C03648=1159.072,-127.448,-41.821,178.641,5.854,149.447
C03649=1159.067,-127.198,-41.829,178.642,5.854,149.447
C03650=1159.061,-126.949,-41.837,178.645,5.855,149.446
C03651=1159.055,-126.699,-41.846,178.646,5.855,149.446
C03652=1159.050,-126.448,-41.854,178.649,5.855,149.445
C03653=1159.045,-126.199,-41.862,178.651,5.855,149.445
C03654=1159.040,-125.950,-41.871,178.653,5.856,149.444
C03655=1159.034,-125.699,-41.879,178.654,5.856,149.444
C03656=1159.029,-125.450,-41.888,178.657,5.856,149.443
C03657=1159.023,-125.200,-41.897,178.659,5.856,149.443
C03658=1159.018,-124.950,-41.906,178.661,5.857,149.442
C03659=1159.013,-124.700,-41.914,178.662,5.857,149.442
C03660=1159.007,-124.451,-41.922,178.665,5.858,149.441
C03661=1159.002,-124.201,-41.931,178.666,5.857,149.441
C03662=1158.996,-123.950,-41.939,178.669,5.858,149.440
C03663=1158.991,-123.701,-41.947,178.670,5.858,149.439
C03664=1158.986,-123.452,-41.956,178.673,5.859,149.439
C03665=1158.981,-123.202,-41.965,178.674,5.859,149.438
C03666=1158.975,-122.952,-41.973,178.676,5.859,149.438
C03667=1158.970,-122.702,-41.982,178.679,5.859,149.437
C03668=1158.965,-122.452,-41.991,178.681,5.860,149.437
C03669=1158.959,-122.202,-42.000,178.682,5.860,149.436
C03670=1158.953,-121.953,-42.008,178.685,5.860,149.436
C03671=1158.948,-121.703,-42.016,178.686,5.860,149.435
C03672=1158.943,-121.453,-42.025,178.689,5.861,149.435
C03673=1158.938,-121.203,-42.034,178.690,5.861,149.434
C03674=1158.932,-120.953,-42.042,178.693,5.861,149.434
C03675=1158.927,-120.703,-42.051,178.694,5.861,149.433
C03676=1158.921,-120.454,-42.060,178.696,5.862,149.433
C03677=1158.916,-120.204,-42.069,178.698,5.862,149.432
C03678=1158.910,-119.955,-42.077,178.701,5.862,149.431
C03679=1158.905,-119.704,-42.085,178.702,5.862,149.431
C03680=1158.900,-119.454,-42.094,178.704,5.863,149.430
C03681=1158.895,-119.204,-42.103,178.707,5.863,149.430
C03682=1158.889,-118.955,-42.112,178.709,5.863,149.429
C03683=1158.884,-118.705,-42.121,178.710,5.863,149.429
C03684=1158.879,-118.456,-42.130,178.713,5.864,149.428
C03685=1158.873,-118.206,-42.138,178.715,5.865,149.428
C03686=1158.868,-117.955,-42.147,178.717,5.865,149.427
C03687=1158.862,-117.706,-42.155,178.719,5.865,149.427
C03688=1158.857,-117.456,-42.164,178.721,5.865,149.426
C03689=1158.852,-117.206,-42.173,178.723,5.866,149.426
C03690=1158.847,-116.957,-42.182,178.725,5.866,149.425
C03691=1158.841,-116.707,-42.190,178.727,5.866,149.424
C03692=1158.836,-116.458,-42.199,178.729,5.866,149.424
C03693=1158.831,-116.208,-42.208,178.731,5.867,149.423
C03694=1158.825,-115.958,-42.217,178.733,5.867,149.423
C03695=1158.820,-115.707,-42.225,178.735,5.867,149.422
C03696=1158.814,-115.458,-42.234,178.737,5.867,149.422
C03697=1158.808,-115.208,-42.243,178.739,5.868,149.421
C03698=1158.803,-114.958,-42.252,178.741,5.868,149.421
C03699=1158.798,-114.708,-42.261,178.743,5.868,149.420
C03700=1158.793,-114.458,-42.270,178.745,5.869,149.420
C03701=1158.788,-114.209,-42.279,178.747,5.869,149.419
C03702=1158.782,-113.959,-42.287,178.750,5.870,149.418
C03703=1158.777,-113.710,-42.296,178.751,5.869,149.418
C03704=1158.771,-113.460,-42.305,178.753,5.870,149.417
C03705=1158.766,-113.210,-42.314,178.755,5.870,149.417
C03706=1158.760,-112.960,-42.324,178.758,5.871,149.416
C03707=1158.755,-112.710,-42.333,178.759,5.871,149.416
C03708=1158.749,-112.461,-42.341,178.762,5.871,149.415
C03709=1158.744,-112.211,-42.350,178.763,5.871,149.415
C03710=1158.739,-111.961,-42.359,178.766,5.872,149.414
C03711=1158.734,-111.711,-42.368,178.768,5.872,149.414
C03712=1158.729,-111.461,-42.377,178.770,5.872,149.413
C03713=1158.723,-111.211,-42.386,178.772,5.873,149.413
C03714=1158.718,-110.961,-42.395,178.774,5.873,149.412
C03715=1158.712,-110.712,-42.404,178.776,5.873,149.411
C03716=1158.707,-110.462,-42.412,178.778,5.873,149.411
C03717=1158.702,-110.213,-42.421,178.780,5.874,149.410
C03718=1158.696,-109.963,-42.430,178.782,5.874,149.410
C03719=1158.691,-109.712,-42.440,178.784,5.875,149.409
C03720=1158.686,-109.463,-42.449,178.786,5.875,149.409
C03721=1158.681,-109.213,-42.458,178.788,5.875,149.408
C03722=1158.675,-108.964,-42.467,178.791,5.876,149.408
C03723=1158.670,-108.714,-42.476,178.792,5.876,149.407
C03724=1158.664,-108.464,-42.485,178.794,5.876,149.407
C03725=1158.659,-108.214,-42.494,178.796,5.876,149.406
C03726=1158.653,-107.965,-42.503,178.799,5.877,149.405
C03727=1158.648,-107.715,-42.512,178.801,5.877,149.405
C03728=1158.643,-107.465,-42.521,178.802,5.877,149.404
C03729=1158.637,-107.215,-42.531,178.805,5.878,149.404
C03730=1158.632,-106.965,-42.540,178.807,5.878,149.403
C03731=1158.627,-106.716,-42.549,178.809,5.879,149.403
C03732=1158.622,-106.466,-42.558,178.811,5.878,149.402
C03733=1158.616,-106.216,-42.567,178.813,5.879,149.401
C03734=1158.611,-105.966,-42.576,178.815,5.880,149.401
C03735=1158.606,-105.716,-42.586,178.817,5.880,149.401
C03736=1158.600,-105.467,-42.594,178.820,5.880,149.400
C03737=1158.594,-105.217,-42.604,178.821,5.880,149.399
C03738=1158.589,-104.967,-42.613,178.823,5.881,149.399
C03739=1158.584,-104.717,-42.622,178.826,5.880,149.398
C03740=1158.579,-104.468,-42.631,178.828,5.881,149.398
C03741=1158.573,-104.218,-42.641,178.830,5.882,149.397
C03742=1158.568,-103.968,-42.650,178.832,5.881,149.396
C03743=1158.563,-103.718,-42.658,178.834,5.882,149.396
C03744=1158.557,-103.469,-42.669,178.836,5.882,149.395
C03745=1158.552,-103.219,-42.678,178.838,5.883,149.395
C03746=1158.547,-102.969,-42.686,178.840,5.882,149.394
C03747=1158.541,-102.697,-42.697,178.842,5.883,149.394
C03748=1158.535,-102.425,-42.707,178.845,5.884,149.393
C03749=1158.529,-102.152,-42.717,178.847,5.884,149.393
C03750=1158.523,-101.881,-42.727,178.849,5.884,149.392
C03751=1158.518,-101.631,-42.736,178.851,5.885,149.391
C03752=1158.513,-101.382,-42.746,178.854,5.885,149.391
C03753=1158.507,-101.132,-42.755,178.856,5.885,149.390
C03754=1158.502,-100.882,-42.764,178.858,5.886,149.390
C03755=1158.497,-100.633,-42.774,178.859,5.886,149.389
C03756=1158.491,-100.383,-42.783,178.862,5.886,149.388
C03757=1158.486,-100.133,-42.792,178.864,5.887,149.388
C03758=1158.481,-99.883,-42.802,178.866,5.887,149.388
C03759=1158.476,-99.633,-42.811,178.869,5.887,149.387
C03760=1158.470,-99.384,-42.820,178.870,5.887,149.386
C03761=1158.465,-99.134,-42.830,178.872,5.888,149.386
C03762=1158.460,-98.884,-42.839,178.875,5.888,149.385
C03763=1158.454,-98.634,-42.848,178.877,5.888,149.385
C03764=1158.449,-98.385,-42.858,178.879,5.889,149.384
C03765=1158.444,-98.135,-42.867,178.881,5.889,149.383
C03766=1158.439,-97.885,-42.877,178.883,5.889,149.383
C03767=1158.434,-97.635,-42.886,178.885,5.890,149.382
C03768=1158.428,-97.385,-42.896,178.887,5.890,149.382
C03769=1158.423,-97.135,-42.905,178.890,5.891,149.381
C03770=1158.417,-96.885,-42.915,178.891,5.891,149.381
C03771=1158.412,-96.636,-42.925,178.893,5.891,149.380
C03772=1158.407,-96.386,-42.933,178.896,5.892,149.380
C03773=1158.401,-96.136,-42.943,178.898,5.892,149.379
C03774=1158.396,-95.887,-42.953,178.900,5.892,149.379
C03775=1158.390,-95.637,-42.962,178.903,5.893,149.378
C03776=1158.385,-95.387,-42.972,178.904,5.893,149.377
C03777=1158.379,-95.137,-42.981,178.906,5.894,149.377
C03778=1158.375,-94.888,-42.991,178.908,5.893,149.376
C03779=1158.369,-94.638,-43.000,178.911,5.894,149.376
C03780=1158.364,-94.389,-43.010,178.913,5.895,149.375
C03781=1158.358,-94.139,-43.019,178.915,5.894,149.375
C03782=1158.354,-93.889,-43.029,178.917,5.895,149.374
C03783=1158.348,-93.638,-43.039,178.920,5.895,149.373
C03784=1158.343,-93.389,-43.048,178.921,5.895,149.373
C03785=1158.337,-93.139,-43.058,178.924,5.896,149.372
C03786=1158.332,-92.890,-43.068,178.926,5.896,149.372
C03787=1158.326,-92.640,-43.077,178.928,5.897,149.371
C03788=1158.321,-92.390,-43.087,178.930,5.897,149.371
C03789=1158.315,-92.140,-43.096,178.932,5.897,149.370
C03790=1158.311,-91.891,-43.106,178.934,5.898,149.370
C03791=1158.305,-91.641,-43.115,178.936,5.898,149.369
C03792=1158.300,-91.391,-43.125,178.939,5.898,149.368
C03793=1158.294,-91.141,-43.135,178.941,5.899,149.368
C03794=1158.290,-90.892,-43.144,178.943,5.900,149.367
C03795=1158.284,-90.642,-43.155,178.945,5.899,149.367
C03796=1158.279,-90.392,-43.163,178.947,5.900,149.366
C03797=1158.273,-90.143,-43.174,178.949,5.900,149.366
C03798=1158.268,-89.893,-43.183,178.951,5.900,149.365
C03799=1158.263,-89.642,-43.193,178.954,5.901,149.364
C03800=1158.257,-89.393,-43.203,178.955,5.901,149.364
C03801=1158.252,-89.143,-43.212,178.958,5.901,149.363
C03802=1158.247,-88.894,-43.222,178.960,5.902,149.363
C03803=1158.242,-88.644,-43.232,178.962,5.902,149.362
C03804=1158.236,-88.394,-43.242,178.964,5.903,149.362
C03805=1158.231,-88.144,-43.252,178.967,5.903,149.361
C03806=1158.226,-87.894,-43.261,178.969,5.903,149.360
C03807=1158.220,-87.645,-43.271,178.971,5.904,149.360
C03808=1158.215,-87.395,-43.281,178.973,5.904,149.359
C03809=1158.209,-87.145,-43.290,178.975,5.904,149.359
C03810=1158.204,-86.896,-43.301,178.977,5.905,149.358
C03811=1158.200,-86.646,-43.311,178.980,5.905,149.358
C03812=1158.194,-86.396,-43.321,178.982,5.905,149.357
C03813=1158.189,-86.146,-43.330,178.984,5.906,149.357
C03814=1158.183,-85.897,-43.340,178.986,5.906,149.356
C03815=1158.178,-85.647,-43.350,178.988,5.906,149.355
C03816=1158.173,-85.397,-43.359,178.990,5.907,149.355
C03817=1158.167,-85.147,-43.370,178.992,5.907,149.354
C03818=1158.162,-84.898,-43.380,178.994,5.907,149.354
C03819=1158.157,-84.648,-43.389,178.997,5.908,149.353
C03820=1158.151,-84.398,-43.399,178.999,5.908,149.353
C03821=1158.146,-84.148,-43.409,179.001,5.909,149.352
C03822=1158.141,-83.899,-43.419,179.004,5.909,149.351
C03823=1158.136,-83.649,-43.429,179.006,5.910,149.351
C03824=1158.130,-83.399,-43.439,179.007,5.910,149.350
C03825=1158.125,-83.149,-43.449,179.010,5.910,149.350
C03826=1158.120,-82.899,-43.459,179.012,5.911,149.349
C03827=1158.114,-82.650,-43.469,179.014,5.910,149.348
C03828=1158.109,-82.400,-43.479,179.017,5.911,149.348
C03829=1158.104,-82.150,-43.489,179.019,5.912,149.348
C03830=1158.099,-81.900,-43.499,179.021,5.912,149.347
C03831=1158.093,-81.651,-43.509,179.023,5.912,149.346
C03832=1158.088,-81.402,-43.519,179.025,5.913,149.346
C03833=1158.083,-81.151,-43.529,179.027,5.913,149.345
C03834=1158.077,-80.902,-43.539,179.029,5.913,149.345
C03835=1158.072,-80.652,-43.550,179.032,5.914,149.344
C03836=1158.067,-80.402,-43.559,179.034,5.914,149.343
C03837=1158.062,-80.152,-43.569,179.036,5.915,149.343
C03838=1158.056,-79.903,-43.579,179.039,5.915,149.342
C03839=1158.050,-79.653,-43.590,179.040,5.915,149.342
C03840=1158.046,-79.403,-43.600,179.043,5.915,149.341
C03841=1158.041,-79.154,-43.610,179.045,5.916,149.341
C03842=1158.035,-78.904,-43.620,179.047,5.916,149.340
C03843=1158.029,-78.654,-43.630,179.049,5.917,149.339
C03844=1158.024,-78.404,-43.641,179.051,5.917,149.339
C03845=1158.019,-78.154,-43.650,179.054,5.918,149.338
C03846=1158.014,-77.905,-43.660,179.056,5.918,149.338
C03847=1158.009,-77.655,-43.670,179.058,5.918,149.337
C03848=1158.003,-77.405,-43.681,179.061,5.919,149.337
C03849=1157.997,-77.155,-43.691,179.062,5.919,149.336
C03850=1157.992,-76.906,-43.701,179.065,5.919,149.335
C03851=1157.987,-76.635,-43.712,179.067,5.920,149.335
C03852=1157.981,-76.363,-43.724,179.070,5.920,149.334
C03853=1157.976,-76.092,-43.734,179.072,5.921,149.334
C03854=1157.969,-75.821,-43.746,179.074,5.921,149.333
C03855=1157.965,-75.571,-43.756,179.076,5.922,149.332
C03856=1157.959,-75.321,-43.766,179.079,5.922,149.332
C03857=1157.954,-75.072,-43.776,179.081,5.923,149.331
C03858=1157.949,-74.822,-43.787,179.083,5.922,149.331
C03859=1157.943,-74.572,-43.797,179.085,5.923,149.330
C03860=1157.937,-74.322,-43.807,179.088,5.923,149.329
C03861=1157.932,-74.072,-43.818,179.090,5.923,149.329
C03862=1157.927,-73.823,-43.828,179.092,5.924,149.328
C03863=1157.921,-73.573,-43.838,179.094,5.925,149.328
C03864=1157.917,-73.323,-43.848,179.097,5.925,149.327
C03865=1157.911,-73.074,-43.858,179.099,5.925,149.327
C03866=1157.906,-72.824,-43.868,179.101,5.926,149.326
C03867=1157.901,-72.574,-43.880,179.103,5.927,149.326
C03868=1157.895,-72.325,-43.890,179.105,5.926,149.325
C03869=1157.890,-72.075,-43.900,179.107,5.927,149.324
C03870=1157.885,-71.825,-43.911,179.110,5.927,149.324
C03871=1157.879,-71.576,-43.921,179.112,5.928,149.323
C03872=1157.874,-71.325,-43.931,179.114,5.928,149.322
C03873=1157.869,-71.076,-43.942,179.117,5.928,149.322
C03874=1157.863,-70.826,-43.952,179.119,5.929,149.322
C03875=1157.858,-70.576,-43.962,179.121,5.930,149.321
C03876=1157.853,-70.327,-43.973,179.123,5.930,149.320
C03877=1157.848,-70.077,-43.984,179.126,5.930,149.320
C03878=1157.842,-69.827,-43.994,179.128,5.931,149.319
C03879=1157.837,-69.577,-44.005,179.131,5.931,149.318
C03880=1157.832,-69.328,-44.015,179.132,5.931,149.318
C03881=1157.826,-69.078,-44.025,179.134,5.932,149.317
C03882=1157.821,-68.828,-44.036,179.137,5.932,149.317
C03883=1157.816,-68.579,-44.047,179.139,5.932,149.316
C03884=1157.811,-68.329,-44.057,179.141,5.933,149.316
C03885=1157.805,-68.079,-44.067,179.143,5.933,149.315
C03886=1157.800,-67.829,-44.078,179.146,5.934,149.314
C03887=1157.795,-67.580,-44.089,179.148,5.934,149.314
C03888=1157.789,-67.330,-44.099,179.150,5.935,149.313
C03889=1157.784,-67.080,-44.110,179.153,5.935,149.313
C03890=1157.779,-66.831,-44.120,179.155,5.936,149.312
C03891=1157.774,-66.581,-44.131,179.157,5.935,149.312
C03892=1157.768,-66.331,-44.141,179.159,5.936,149.311
C03893=1157.763,-66.081,-44.152,179.162,5.937,149.310
C03894=1157.758,-65.832,-44.162,179.164,5.937,149.310
C03895=1157.753,-65.582,-44.173,179.165,5.937,149.309
C03896=1157.747,-65.332,-44.184,179.168,5.938,149.309
C03897=1157.742,-65.082,-44.194,179.170,5.939,149.308
C03898=1157.737,-64.833,-44.205,179.173,5.939,149.307
C03899=1157.732,-64.583,-44.216,179.175,5.940,149.307
C03900=1157.727,-64.333,-44.226,179.177,5.939,149.306
C03901=1157.722,-64.084,-44.237,179.179,5.940,149.306
C03902=1157.716,-63.834,-44.247,179.182,5.941,149.305
C03903=1157.711,-63.584,-44.258,179.184,5.941,149.305
C03904=1157.705,-63.335,-44.270,179.186,5.941,149.304
C03905=1157.700,-63.085,-44.280,179.189,5.942,149.303
C03906=1157.695,-62.835,-44.290,179.191,5.942,149.303
C03907=1157.690,-62.585,-44.302,179.193,5.943,149.302
C03908=1157.684,-62.336,-44.312,179.195,5.943,149.302
C03909=1157.679,-62.086,-44.322,179.198,5.943,149.301
C03910=1157.674,-61.837,-44.333,179.200,5.944,149.301
C03911=1157.669,-61.586,-44.344,179.203,5.944,149.300
C03912=1157.663,-61.337,-44.355,179.205,5.945,149.299
C03913=1157.658,-61.087,-44.366,179.206,5.945,149.299
C03914=1157.652,-60.837,-44.376,179.209,5.946,149.298
C03915=1157.648,-60.588,-44.388,179.211,5.946,149.298
C03916=1157.643,-60.338,-44.398,179.214,5.947,149.297
C03917=1157.637,-60.089,-44.409,179.215,5.947,149.297
C03918=1157.632,-59.838,-44.420,179.218,5.947,149.296
C03919=1157.626,-59.589,-44.431,179.220,5.948,149.295
C03920=1157.621,-59.339,-44.442,179.223,5.948,149.295
C03921=1157.616,-59.090,-44.453,179.225,5.949,149.294
C03922=1157.611,-58.840,-44.463,179.227,5.949,149.294
C03923=1157.606,-58.590,-44.474,179.229,5.950,149.293
C03924=1157.600,-58.340,-44.485,179.232,5.950,149.293
C03925=1157.595,-58.091,-44.497,179.234,5.951,149.292
C03926=1157.590,-57.841,-44.507,179.236,5.952,149.291
C03927=1157.585,-57.591,-44.518,179.238,5.951,149.291
C03928=1157.580,-57.341,-44.529,179.241,5.952,149.290
C03929=1157.574,-57.092,-44.540,179.243,5.952,149.289
C03930=1157.569,-56.842,-44.551,179.246,5.953,149.289
C03931=1157.564,-56.593,-44.562,179.248,5.954,149.288
C03932=1157.559,-56.343,-44.572,179.250,5.954,149.288
C03933=1157.553,-56.093,-44.584,179.252,5.954,149.287
C03934=1157.548,-55.844,-44.595,179.255,5.955,149.287
C03935=1157.543,-55.593,-44.606,179.257,5.955,149.286
C03936=1157.538,-55.345,-44.617,179.260,5.956,149.285
C03937=1157.532,-55.094,-44.628,179.261,5.956,149.285
C03938=1157.527,-54.844,-44.639,179.264,5.956,149.284
C03939=1157.522,-54.595,-44.649,179.266,5.957,149.284
C03940=1157.517,-54.345,-44.661,179.269,5.957,149.283
C03941=1157.512,-54.095,-44.672,179.271,5.958,149.283
C03942=1157.506,-53.846,-44.683,179.273,5.958,149.282
C03943=1157.501,-53.596,-44.694,179.275,5.959,149.281
C03944=1157.496,-53.346,-44.706,179.278,5.959,149.281
C03945=1157.490,-53.097,-44.716,179.280,5.960,149.280
C03946=1157.486,-52.847,-44.727,179.283,5.960,149.280
C03947=1157.480,-52.597,-44.739,179.284,5.960,149.279
C03948=1157.475,-52.347,-44.749,179.287,5.961,149.278
C03949=1157.470,-52.098,-44.761,179.289,5.961,149.278
C03950=1157.465,-51.848,-44.773,179.292,5.962,149.277
C03951=1157.459,-51.598,-44.783,179.294,5.963,149.277
C03952=1157.454,-51.349,-44.794,179.296,5.963,149.276
C03953=1157.449,-51.099,-44.806,179.298,5.963,149.276
C03954=1157.443,-50.849,-44.816,179.300,5.964,149.275
C03955=1157.438,-50.579,-44.829,179.303,5.964,149.274
C03956=1157.432,-50.308,-44.841,179.306,5.965,149.274
C03957=1157.426,-50.038,-44.853,179.308,5.965,149.273
C03958=1157.421,-49.767,-44.865,179.311,5.966,149.272
C03959=1157.416,-49.517,-44.877,179.313,5.966,149.272
C03960=1157.410,-49.268,-44.888,179.315,5.967,149.271
C03961=1157.405,-49.018,-44.899,179.318,5.967,149.271
C03962=1157.400,-48.768,-44.910,179.320,5.968,149.270
C03963=1157.395,-48.519,-44.921,179.322,5.968,149.269
C03964=1157.389,-48.269,-44.933,179.324,5.969,149.269
C03965=1157.385,-48.019,-44.944,179.327,5.969,149.268
C03966=1157.379,-47.769,-44.955,179.329,5.970,149.268
C03967=1157.374,-47.520,-44.966,179.332,5.971,149.267
C03968=1157.368,-47.270,-44.978,179.334,5.971,149.267
C03969=1157.363,-47.020,-44.990,179.336,5.971,149.266
C03970=1157.357,-46.771,-45.001,179.338,5.971,149.265
C03971=1157.353,-46.522,-45.012,179.341,5.972,149.265
C03972=1157.347,-46.271,-45.024,179.343,5.973,149.264
C03973=1157.342,-46.021,-45.035,179.345,5.973,149.264
C03974=1157.338,-45.772,-45.046,179.348,5.974,149.263
C03975=1157.332,-45.523,-45.058,179.350,5.975,149.263
C03976=1157.327,-45.273,-45.069,179.352,5.974,149.262
C03977=1157.321,-45.023,-45.081,179.355,5.975,149.261
C03978=1157.317,-44.773,-45.092,179.357,5.975,149.261
C03979=1157.311,-44.524,-45.104,179.359,5.976,149.260
C03980=1157.306,-44.274,-45.115,179.362,5.977,149.259
C03981=1157.301,-44.025,-45.127,179.364,5.977,149.259
C03982=1157.296,-43.774,-45.137,179.367,5.978,149.258
C03983=1157.290,-43.524,-45.149,179.369,5.979,149.258
C03984=1157.284,-43.275,-45.161,179.371,5.978,149.257
C03985=1157.279,-43.025,-45.172,179.373,5.979,149.257
C03986=1157.274,-42.776,-45.184,179.376,5.979,149.256
C03987=1157.269,-42.526,-45.195,179.378,5.980,149.255
C03988=1157.264,-42.276,-45.207,179.381,5.981,149.255
C03989=1157.259,-42.027,-45.218,179.383,5.981,149.254
C03990=1157.253,-41.777,-45.230,179.386,5.982,149.254
C03991=1157.248,-41.528,-45.241,179.388,5.983,149.253
C03992=1157.243,-41.278,-45.253,179.390,5.982,149.252
C03993=1157.238,-41.028,-45.265,179.392,5.983,149.252
C03994=1157.232,-40.779,-45.276,179.395,5.984,149.251
C03995=1157.227,-40.529,-45.288,179.397,5.984,149.251
C03996=1157.222,-40.279,-45.299,179.400,5.985,149.250
C03997=1157.217,-40.029,-45.311,179.402,5.986,149.250
C03998=1157.211,-39.779,-45.323,179.405,5.986,149.249
C03999=1157.207,-39.530,-45.334,179.407,5.987,149.248
C04000=1157.202,-39.280,-45.347,179.409,5.986,149.248
C04001=1157.196,-39.031,-45.358,179.411,5.987,149.247
C04002=1157.191,-38.781,-45.370,179.413,5.988,149.247
C04003=1157.185,-38.532,-45.381,179.416,5.988,149.246
C04004=1157.181,-38.282,-45.393,179.418,5.989,149.246
C04005=1157.175,-38.032,-45.405,179.421,5.990,149.245
C04006=1157.170,-37.782,-45.416,179.423,5.990,149.244
C04007=1157.165,-37.532,-45.428,179.426,5.991,149.244
C04008=1157.159,-37.283,-45.439,179.428,5.992,149.243
C04009=1157.154,-37.033,-45.451,179.430,5.992,149.243
C04010=1157.149,-36.784,-45.463,179.432,5.992,149.242
C04011=1157.144,-36.534,-45.475,179.435,5.992,149.241
C04012=1157.138,-36.284,-45.487,179.437,5.993,149.241
C04013=1157.134,-36.035,-45.498,179.439,5.994,149.240
C04014=1157.128,-35.785,-45.510,179.442,5.994,149.240
C04015=1157.123,-35.535,-45.522,179.444,5.995,149.239
C04016=1157.119,-35.286,-45.534,179.447,5.996,149.239
C04017=1157.113,-35.036,-45.546,179.449,5.996,149.238
C04018=1157.107,-34.787,-45.557,179.451,5.997,149.237
C04019=1157.102,-34.537,-45.569,179.454,5.997,149.237
C04020=1157.097,-34.288,-45.581,179.456,5.998,149.236
C04021=1157.092,-34.038,-45.593,179.458,5.998,149.236
C04022=1157.086,-33.788,-45.605,179.460,5.999,149.235
C04023=1157.081,-33.538,-45.617,179.463,5.999,149.234
C04024=1157.077,-33.289,-45.629,179.465,6.000,149.234
C04025=1157.071,-33.039,-45.641,179.468,6.000,149.233
C04026=1157.066,-32.789,-45.653,179.470,6.001,149.233
C04027=1157.060,-32.539,-45.665,179.473,6.001,149.232
C04028=1157.056,-32.290,-45.677,179.475,6.002,149.232
C04029=1157.050,-32.040,-45.689,179.478,6.003,149.231
C04030=1157.045,-31.790,-45.700,179.480,6.003,149.230
C04031=1157.040,-31.541,-45.713,179.483,6.004,149.230
C04032=1157.034,-31.291,-45.725,179.485,6.005,149.229
C04033=1157.030,-31.041,-45.736,179.487,6.005,149.228
C04034=1157.024,-30.791,-45.748,179.490,6.006,149.228
C04035=1157.019,-30.542,-45.761,179.492,6.005,149.227
C04036=1157.014,-30.292,-45.773,179.494,6.006,149.227
C04037=1157.009,-30.043,-45.785,179.496,6.007,149.226
C04038=1157.004,-29.793,-45.796,179.499,6.007,149.225
C04039=1156.999,-29.543,-45.808,179.501,6.008,149.225
C04040=1156.993,-29.294,-45.821,179.504,6.008,149.224
C04041=1156.988,-29.044,-45.833,179.506,6.009,149.224
C04042=1156.983,-28.794,-45.845,179.509,6.010,149.223
C04043=1156.977,-28.545,-45.857,179.511,6.010,149.223
C04044=1156.972,-28.295,-45.869,179.514,6.011,149.222
C04045=1156.968,-28.046,-45.881,179.516,6.012,149.221
C04046=1156.962,-27.796,-45.893,179.518,6.012,149.221
C04047=1156.957,-27.547,-45.906,179.521,6.013,149.220
C04048=1156.952,-27.297,-45.918,179.523,6.013,149.220
C04049=1156.946,-27.047,-45.929,179.526,6.014,149.219
C04050=1156.941,-26.797,-45.942,179.528,6.014,149.218
C04051=1156.936,-26.547,-45.954,179.530,6.015,149.218
C04052=1156.931,-26.298,-45.967,179.533,6.016,149.217
C04053=1156.926,-26.049,-45.978,179.535,6.016,149.217
C04054=1156.921,-25.799,-45.990,179.538,6.017,149.216
C04055=1156.915,-25.549,-46.002,179.540,6.018,149.216
C04056=1156.910,-25.300,-46.015,179.543,6.018,149.215
C04057=1156.905,-25.050,-46.027,179.544,6.018,149.214
C04058=1156.900,-24.800,-46.040,179.547,6.019,149.214
C04059=1156.894,-24.530,-46.052,179.550,6.020,149.213
C04060=1156.889,-24.260,-46.067,179.552,6.021,149.213
C04061=1156.883,-23.991,-46.079,179.555,6.021,149.212
C04062=1156.878,-23.721,-46.093,179.558,6.021,149.211
C04063=1156.872,-23.471,-46.105,179.560,6.022,149.211
C04064=1156.867,-23.222,-46.117,179.563,6.023,149.210
C04065=1156.862,-22.972,-46.129,179.565,6.023,149.210
C04066=1156.857,-22.722,-46.142,179.567,6.024,149.209
C04067=1156.852,-22.472,-46.154,179.570,6.025,149.208
C04068=1156.847,-22.222,-46.167,179.572,6.025,149.208
C04069=1156.841,-21.973,-46.179,179.574,6.026,149.207
C04070=1156.836,-21.723,-46.191,179.577,6.026,149.207
C04071=1156.831,-21.474,-46.204,179.579,6.027,149.206
C04072=1156.826,-21.225,-46.216,179.582,6.028,149.205
C04073=1156.820,-20.975,-46.228,179.584,6.028,149.205
C04074=1156.815,-20.725,-46.241,179.587,6.029,149.204
C04075=1156.811,-20.475,-46.254,179.589,6.030,149.204
C04076=1156.805,-20.225,-46.266,179.592,6.030,149.203
C04077=1156.800,-19.976,-46.278,179.594,6.031,149.203
C04078=1156.794,-19.726,-46.292,179.596,6.031,149.202
C04079=1156.789,-19.476,-46.303,179.599,6.032,149.201
C04080=1156.784,-19.227,-46.316,179.601,6.033,149.201
C04081=1156.779,-18.978,-46.329,179.603,6.033,149.200
C04082=1156.774,-18.727,-46.341,179.606,6.034,149.200
C04083=1156.769,-18.478,-46.354,179.608,6.035,149.199
C04084=1156.764,-18.229,-46.366,179.611,6.035,149.198
C04085=1156.758,-17.979,-46.379,179.613,6.036,149.198
C04086=1156.753,-17.729,-46.391,179.616,6.036,149.197
C04087=1156.748,-17.479,-46.404,179.618,6.037,149.197
C04088=1156.743,-17.230,-46.416,179.621,6.037,149.196
C04089=1156.737,-16.980,-46.429,179.623,6.038,149.196
C04090=1156.732,-16.730,-46.441,179.625,6.039,149.195
C04091=1156.727,-16.481,-46.454,179.628,6.040,149.194
C04092=1156.722,-16.231,-46.467,179.630,6.040,149.194
C04093=1156.717,-15.982,-46.479,179.632,6.041,149.193
C04094=1156.712,-15.732,-46.492,179.635,6.041,149.193
C04095=1156.707,-15.482,-46.504,179.637,6.042,149.192
C04096=1156.701,-15.233,-46.517,179.640,6.042,149.191
C04097=1156.696,-14.983,-46.530,179.642,6.043,149.191
C04098=1156.691,-14.734,-46.543,179.645,6.044,149.190
C04099=1156.686,-14.484,-46.555,179.647,6.044,149.190
C04100=1156.681,-14.235,-46.568,179.650,6.045,149.189
C04101=1156.676,-13.985,-46.581,179.652,6.045,149.188
C04102=1156.670,-13.735,-46.593,179.655,6.046,149.188
C04103=1156.665,-13.485,-46.606,179.657,6.047,149.187
C04104=1156.660,-13.236,-46.619,179.659,6.047,149.187
C04105=1156.656,-12.986,-46.631,179.662,6.048,149.186
C04106=1156.650,-12.736,-46.645,179.664,6.049,149.186
C04107=1156.645,-12.487,-46.657,179.667,6.049,149.185
C04108=1156.639,-12.238,-46.670,179.669,6.050,149.184
C04109=1156.635,-11.988,-46.683,179.672,6.050,149.184
C04110=1156.630,-11.738,-46.695,179.674,6.051,149.183
C04111=1156.624,-11.489,-46.709,179.677,6.052,149.183
C04112=1156.619,-11.239,-46.721,179.679,6.053,149.182
C04113=1156.614,-10.989,-46.734,179.682,6.054,149.181
C04114=1156.609,-10.740,-46.747,179.684,6.054,149.181
C04115=1156.603,-10.490,-46.760,179.687,6.055,149.180
C04116=1156.599,-10.240,-46.773,179.689,6.056,149.180
C04117=1156.594,-9.991,-46.786,179.692,6.056,149.179
C04118=1156.588,-9.741,-46.799,179.694,6.057,149.179
C04119=1156.583,-9.491,-46.812,179.696,6.057,149.178
C04120=1156.578,-9.242,-46.824,179.699,6.058,149.177
C04121=1156.573,-8.993,-46.837,179.701,6.059,149.177
C04122=1156.568,-8.742,-46.850,179.703,6.059,149.176
C04123=1156.563,-8.493,-46.863,179.706,6.060,149.176
C04124=1156.557,-8.244,-46.876,179.708,6.061,149.175
C04125=1156.552,-7.994,-46.889,179.711,6.061,149.174
C04126=1156.547,-7.744,-46.902,179.713,6.062,149.174
C04127=1156.542,-7.495,-46.914,179.716,6.062,149.173
C04128=1156.537,-7.245,-46.928,179.719,6.064,149.173
C04129=1156.532,-6.995,-46.941,179.721,6.064,149.172
C04130=1156.527,-6.747,-46.954,179.723,6.065,149.172
C04131=1156.522,-6.496,-46.967,179.726,6.066,149.171
C04132=1156.516,-6.247,-46.980,179.729,6.066,149.170
C04133=1156.511,-5.997,-46.993,179.731,6.067,149.170
C04134=1156.506,-5.747,-47.006,179.734,6.067,149.169
C04135=1156.501,-5.498,-47.019,179.736,6.068,149.169
C04136=1156.496,-5.248,-47.032,179.738,6.069,149.168
C04137=1156.491,-4.999,-47.046,179.741,6.070,149.168
C04138=1156.485,-4.749,-47.059,179.743,6.070,149.167
C04139=1156.480,-4.499,-47.072,179.745,6.071,149.166
C04140=1156.475,-4.250,-47.084,179.748,6.071,149.166
C04141=1156.469,-4.000,-47.098,179.751,6.073,149.165
C04142=1156.465,-3.751,-47.111,179.753,6.073,149.165
C04143=1156.459,-3.501,-47.125,179.756,6.074,149.164
C04144=1156.455,-3.251,-47.138,179.758,6.075,149.163
C04145=1156.449,-3.002,-47.151,179.760,6.075,149.163
C04146=1156.445,-2.752,-47.164,179.763,6.076,149.162
C04147=1156.440,-2.503,-47.177,179.765,6.077,149.162
C04148=1156.434,-2.253,-47.190,179.768,6.077,149.161
C04149=1156.429,-2.003,-47.203,179.770,6.078,149.161
C04150=1156.424,-1.754,-47.217,179.773,6.078,149.160
C04151=1156.419,-1.504,-47.230,179.776,6.080,149.159
C04152=1156.413,-1.255,-47.243,179.778,6.080,149.159
C04153=1156.409,-1.005,-47.257,179.780,6.081,149.158
C04154=1156.403,-0.756,-47.270,179.783,6.082,149.158
C04155=1156.398,-0.506,-47.283,179.785,6.082,149.157
C04156=1156.393,-0.257,-47.297,179.788,6.083,149.156
C04157=1156.388,-0.007,-47.310,179.790,6.084,149.156
C04158=1156.383,0.243,-47.323,179.793,6.084,149.155
C04159=1156.377,0.492,-47.337,179.795,6.085,149.155
C04160=1156.373,0.742,-47.350,179.798,6.086,149.154
C04161=1156.367,0.992,-47.363,179.800,6.087,149.154
C04162=1156.363,1.241,-47.377,179.803,6.087,149.153
C04163=1156.356,1.510,-47.391,179.806,6.088,149.152
C04164=1156.351,1.780,-47.406,179.808,6.089,149.152
C04165=1156.346,2.049,-47.420,179.811,6.090,149.151
C04166=1156.340,2.319,-47.435,179.814,6.090,149.150
C04167=1156.335,2.568,-47.448,179.816,6.091,149.150
C04168=1156.330,2.818,-47.461,179.818,6.092,149.149
C04169=1156.324,3.068,-47.475,179.821,6.093,149.149
C04170=1156.320,3.317,-47.489,179.823,6.093,149.148
C04171=1156.314,3.567,-47.501,179.826,6.095,149.148
C04172=1156.309,3.816,-47.516,179.829,6.095,149.147
C04173=1156.304,4.066,-47.528,179.831,6.096,149.147
C04174=1156.299,4.315,-47.543,179.834,6.096,149.146
C04175=1156.293,4.565,-47.556,179.836,6.097,149.145
C04176=1156.289,4.814,-47.569,179.838,6.098,149.145
C04177=1156.283,5.064,-47.583,179.841,6.098,149.144
C04178=1156.278,5.314,-47.597,179.844,6.100,149.144
C04179=1156.273,5.563,-47.610,179.846,6.100,149.143
C04180=1156.268,5.813,-47.624,179.849,6.101,149.142
C04181=1156.264,6.062,-47.638,179.851,6.102,149.142
C04182=1156.258,6.312,-47.651,179.853,6.102,149.141
C04183=1156.253,6.562,-47.665,179.856,6.103,149.141
C04184=1156.247,6.811,-47.678,179.858,6.103,149.140
C04185=1156.243,7.061,-47.692,179.862,6.105,149.139
C04186=1156.237,7.310,-47.705,179.864,6.106,149.139
C04187=1156.232,7.560,-47.719,179.866,6.106,149.138
C04188=1156.228,7.809,-47.733,179.869,6.107,149.138
C04189=1156.222,8.059,-47.746,179.871,6.107,149.137
C04190=1156.217,8.309,-47.760,179.873,6.108,149.137
C04191=1156.212,8.558,-47.773,179.877,6.109,149.136
C04192=1156.207,8.808,-47.787,179.879,6.110,149.136
C04193=1156.202,9.057,-47.802,179.881,6.111,149.135
C04194=1156.197,9.307,-47.815,179.884,6.111,149.134
C04195=1156.192,9.556,-47.829,179.886,6.112,149.134
C04196=1156.187,9.805,-47.842,179.888,6.113,149.133
C04197=1156.181,10.056,-47.856,179.892,6.114,149.133
C04198=1156.177,10.306,-47.870,179.894,6.115,149.132
C04199=1156.171,10.555,-47.884,179.896,6.115,149.131
C04200=1156.167,10.804,-47.898,179.899,6.116,149.131
C04201=1156.161,11.054,-47.911,179.901,6.117,149.130
C04202=1156.156,11.303,-47.925,179.904,6.118,149.130
C04203=1156.151,11.553,-47.940,179.907,6.119,149.129
C04204=1156.146,11.803,-47.953,179.909,6.119,149.129
C04205=1156.141,12.052,-47.967,179.912,6.120,149.128
C04206=1156.136,12.302,-47.981,179.914,6.121,149.128
C04207=1156.131,12.551,-47.995,179.916,6.121,149.127
C04208=1156.125,12.800,-48.009,179.919,6.123,149.126
C04209=1156.120,13.051,-48.023,179.922,6.123,149.126
C04210=1156.116,13.300,-48.036,179.924,6.124,149.125
C04211=1156.110,13.549,-48.050,179.927,6.125,149.125
C04212=1156.105,13.799,-48.064,179.929,6.125,149.124
C04213=1156.101,14.049,-48.079,179.932,6.127,149.123
C04214=1156.095,14.298,-48.092,179.934,6.127,149.123
C04215=1156.090,14.548,-48.106,179.937,6.128,149.122
C04216=1156.085,14.798,-48.120,179.939,6.129,149.122
C04217=1156.079,15.047,-48.134,179.942,6.129,149.121
C04218=1156.075,15.296,-48.148,179.944,6.131,149.121
C04219=1156.070,15.546,-48.162,179.947,6.131,149.120
C04220=1156.065,15.795,-48.177,179.949,6.132,149.120
C04221=1156.059,16.044,-48.190,179.952,6.133,149.119
C04222=1156.054,16.295,-48.204,179.954,6.133,149.118
C04223=1156.049,16.545,-48.218,179.957,6.135,149.118
C04224=1156.044,16.794,-48.232,179.959,6.136,149.117
C04225=1156.039,17.043,-48.247,179.962,6.136,149.117
C04226=1156.034,17.293,-48.261,179.964,6.137,149.116
C04227=1156.029,17.543,-48.275,179.968,6.138,149.115
C04228=1156.023,17.792,-48.289,179.970,6.139,149.115
C04229=1156.018,18.041,-48.303,179.972,6.139,149.114
C04230=1156.013,18.291,-48.318,179.975,6.140,149.114
C04231=1156.008,18.541,-48.332,179.977,6.141,149.113
C04232=1156.003,18.791,-48.346,179.980,6.142,149.113
C04233=1155.998,19.040,-48.360,179.983,6.143,149.112
C04234=1155.993,19.289,-48.374,179.985,6.144,149.112
C04235=1155.988,19.539,-48.389,179.987,6.144,149.111
C04236=1155.983,19.789,-48.403,179.990,6.146,149.110
C04237=1155.978,20.038,-48.417,179.993,6.146,149.110
C04238=1155.973,20.287,-48.431,179.995,6.147,149.109
C04239=1155.968,20.537,-48.445,179.998,6.147,149.109
C04240=1155.963,20.787,-48.460,-180.000,6.149,149.108
C04241=1155.958,21.037,-48.474,-179.997,6.149,149.107
C04242=1155.952,21.286,-48.488,-179.995,6.150,149.107
C04243=1155.947,21.535,-48.502,-179.992,6.151,149.106
C04244=1155.943,21.784,-48.517,-179.989,6.152,149.106
C04245=1155.938,22.034,-48.531,-179.987,6.153,149.105
C04246=1155.933,22.284,-48.546,-179.985,6.154,149.105
C04247=1155.928,22.533,-48.560,-179.982,6.154,149.104
C04248=1155.922,22.782,-48.574,-179.979,6.156,149.104
C04249=1155.917,23.032,-48.588,-179.977,6.156,149.103
C04250=1155.912,23.282,-48.602,-179.974,6.157,149.102
C04251=1155.907,23.532,-48.617,-179.972,6.158,149.102
C04252=1155.903,23.781,-48.632,-179.969,6.159,149.101
C04253=1155.897,24.031,-48.646,-179.966,6.160,149.101
C04254=1155.891,24.280,-48.660,-179.964,6.161,149.100
C04255=1155.886,24.529,-48.675,-179.961,6.161,149.100
C04256=1155.881,24.779,-48.689,-179.959,6.163,149.099
C04257=1155.877,25.028,-48.704,-179.956,6.163,149.098
C04258=1155.872,25.278,-48.718,-179.954,6.164,149.098
C04259=1155.867,25.528,-48.732,-179.951,6.164,149.097
C04260=1155.861,25.778,-48.747,-179.948,6.166,149.097
C04261=1155.857,26.027,-48.762,-179.946,6.166,149.096
C04262=1155.851,26.276,-48.776,-179.944,6.167,149.096
C04263=1155.846,26.525,-48.791,-179.941,6.169,149.095
C04264=1155.841,26.775,-48.805,-179.938,6.169,149.095
C04265=1155.836,27.024,-48.820,-179.936,6.170,149.094
C04266=1155.831,27.274,-48.835,-179.933,6.171,149.093
C04267=1155.826,27.543,-48.850,-179.930,6.172,149.093
C04268=1155.820,27.812,-48.866,-179.928,6.173,149.092
C04269=1155.815,28.081,-48.881,-179.925,6.174,149.092
C04270=1155.809,28.350,-48.897,-179.922,6.175,149.091
C04271=1155.805,28.599,-48.912,-179.919,6.176,149.090
C04272=1155.800,28.849,-48.927,-179.917,6.177,149.090
C04273=1155.795,29.099,-48.941,-179.915,6.178,149.089
C04274=1155.789,29.348,-48.956,-179.912,6.178,149.089
C04275=1155.784,29.597,-48.970,-179.909,6.180,149.088
C04276=1155.779,29.847,-48.985,-179.907,6.180,149.088
C04277=1155.773,30.096,-49.000,-179.904,6.181,149.087
C04278=1155.768,30.346,-49.015,-179.902,6.183,149.087
C04279=1155.764,30.595,-49.030,-179.899,6.183,149.086
C04280=1155.759,30.845,-49.044,-179.897,6.184,149.086
C04281=1155.753,31.094,-49.059,-179.894,6.185,149.085
C04282=1155.748,31.344,-49.074,-179.891,6.186,149.084
C04283=1155.743,31.594,-49.088,-179.889,6.186,149.084
C04284=1155.738,31.843,-49.104,-179.887,6.187,149.083
C04285=1155.733,32.093,-49.118,-179.883,6.189,149.083
C04286=1155.728,32.342,-49.133,-179.881,6.189,149.082
C04287=1155.724,32.592,-49.147,-179.879,6.190,149.081
C04288=1155.718,32.841,-49.163,-179.876,6.192,149.081
C04289=1155.713,33.091,-49.177,-179.873,6.192,149.080
C04290=1155.709,33.340,-49.192,-179.871,6.193,149.080
C04291=1155.703,33.590,-49.207,-179.868,6.194,149.079
C04292=1155.698,33.839,-49.222,-179.866,6.195,149.079
C04293=1155.693,34.089,-49.237,-179.863,6.195,149.078
C04294=1155.688,34.338,-49.252,-179.860,6.197,149.078
C04295=1155.683,34.587,-49.267,-179.858,6.198,149.077
C04296=1155.678,34.837,-49.282,-179.855,6.198,149.076
C04297=1155.673,35.086,-49.297,-179.853,6.200,149.076
C04298=1155.667,35.336,-49.311,-179.850,6.200,149.075
C04299=1155.663,35.585,-49.326,-179.848,6.201,149.075
C04300=1155.658,35.835,-49.341,-179.845,6.203,149.074
C04301=1155.653,36.085,-49.357,-179.842,6.203,149.074
C04302=1155.648,36.334,-49.372,-179.840,6.204,149.073
C04303=1155.642,36.584,-49.387,-179.837,6.206,149.073
C04304=1155.638,36.833,-49.402,-179.834,6.206,149.072
C04305=1155.632,37.083,-49.417,-179.832,6.207,149.072
C04306=1155.627,37.333,-49.431,-179.829,6.208,149.071
C04307=1155.623,37.582,-49.446,-179.827,6.209,149.070
C04308=1155.617,37.831,-49.462,-179.824,6.209,149.070
C04309=1155.612,38.081,-49.476,-179.821,6.211,149.069
C04310=1155.607,38.330,-49.492,-179.819,6.212,149.069
C04311=1155.602,38.579,-49.507,-179.817,6.212,149.068
C04312=1155.597,38.829,-49.522,-179.814,6.214,149.068
C04313=1155.592,39.078,-49.537,-179.811,6.215,149.067
C04314=1155.587,39.328,-49.553,-179.808,6.216,149.067
C04315=1155.583,39.578,-49.568,-179.806,6.217,149.066
C04316=1155.577,39.828,-49.583,-179.804,6.218,149.065
C04317=1155.572,40.077,-49.598,-179.800,6.219,149.065
C04318=1155.567,40.326,-49.613,-179.798,6.220,149.064
C04319=1155.562,40.575,-49.628,-179.796,6.220,149.064
C04320=1155.557,40.825,-49.644,-179.793,6.222,149.063
C04321=1155.551,41.075,-49.659,-179.790,6.222,149.063
C04322=1155.547,41.324,-49.674,-179.787,6.224,149.062
C04323=1155.542,41.574,-49.689,-179.785,6.224,149.061
C04324=1155.537,41.823,-49.704,-179.783,6.225,149.061
C04325=1155.532,42.072,-49.720,-179.780,6.227,149.061
C04326=1155.527,42.322,-49.734,-179.777,6.227,149.060
C04327=1155.521,42.571,-49.750,-179.775,6.228,149.059
C04328=1155.517,42.821,-49.766,-179.772,6.229,149.059
C04329=1155.512,43.071,-49.781,-179.770,6.230,149.058
C04330=1155.507,43.320,-49.796,-179.766,6.232,149.058
C04331=1155.502,43.569,-49.811,-179.764,6.232,149.057
C04332=1155.497,43.818,-49.827,-179.762,6.233,149.057
C04333=1155.492,44.069,-49.843,-179.759,6.235,149.056
C04334=1155.487,44.318,-49.858,-179.757,6.235,149.056
C04335=1155.482,44.567,-49.874,-179.754,6.237,149.055
C04336=1155.476,44.817,-49.888,-179.751,6.238,149.055
C04337=1155.471,45.066,-49.903,-179.749,6.238,149.054
C04338=1155.467,45.316,-49.919,-179.746,6.240,149.053
C04339=1155.462,45.565,-49.934,-179.743,6.240,149.053
C04340=1155.457,45.815,-49.950,-179.741,6.242,149.052
C04341=1155.451,46.064,-49.966,-179.738,6.242,149.052
C04342=1155.447,46.313,-49.981,-179.736,6.243,149.051
C04343=1155.442,46.563,-49.997,-179.733,6.245,149.051
C04344=1155.436,46.813,-50.012,-179.730,6.245,149.050
C04345=1155.431,47.062,-50.028,-179.728,6.247,149.050
C04346=1155.426,47.311,-50.043,-179.725,6.247,149.049
C04347=1155.422,47.561,-50.059,-179.723,6.248,149.049
C04348=1155.416,47.811,-50.074,-179.720,6.250,149.048
C04349=1155.412,48.059,-50.090,-179.717,6.250,149.047
C04350=1155.407,48.309,-50.106,-179.714,6.252,149.047
C04351=1155.402,48.559,-50.121,-179.712,6.253,149.046
C04352=1155.396,48.808,-50.137,-179.710,6.253,149.046
C04353=1155.392,49.057,-50.152,-179.707,6.255,149.045
C04354=1155.387,49.307,-50.168,-179.705,6.256,149.045
C04355=1155.381,49.557,-50.184,-179.701,6.257,149.044
C04356=1155.376,49.806,-50.199,-179.699,6.258,149.044
C04357=1155.372,50.056,-50.215,-179.696,6.259,149.043
C04358=1155.367,50.305,-50.231,-179.694,6.260,149.043
C04359=1155.361,50.554,-50.246,-179.692,6.261,149.042
C04360=1155.357,50.804,-50.262,-179.688,6.262,149.041
C04361=1155.351,51.054,-50.278,-179.686,6.263,149.041
C04362=1155.347,51.303,-50.293,-179.683,6.264,149.040
C04363=1155.341,51.552,-50.309,-179.681,6.265,149.040
C04364=1155.337,51.802,-50.325,-179.678,6.266,149.039
C04365=1155.331,52.051,-50.341,-179.675,6.267,149.039
C04366=1155.327,52.301,-50.357,-179.673,6.269,149.038
C04367=1155.321,52.551,-50.372,-179.670,6.269,149.038
C04368=1155.317,52.799,-50.388,-179.668,6.270,149.037
C04369=1155.312,53.049,-50.404,-179.665,6.271,149.037
C04370=1155.307,53.299,-50.420,-179.663,6.272,149.036
C04371=1155.301,53.567,-50.437,-179.659,6.274,149.035
C04372=1155.296,53.835,-50.454,-179.657,6.275,149.035
C04373=1155.290,54.104,-50.471,-179.654,6.276,149.034
C04374=1155.285,54.373,-50.488,-179.651,6.277,149.034
C04375=1155.280,54.623,-50.504,-179.649,6.278,149.033
C04376=1155.275,54.871,-50.520,-179.646,6.280,149.033
C04377=1155.270,55.121,-50.536,-179.643,6.280,149.032
C04378=1155.264,55.371,-50.551,-179.640,6.282,149.032
C04379=1155.260,55.620,-50.568,-179.638,6.282,149.031
C04380=1155.255,55.869,-50.583,-179.635,6.284,149.031
C04381=1155.250,56.118,-50.599,-179.632,6.284,149.030
C04382=1155.245,56.368,-50.615,-179.630,6.286,149.029
C04383=1155.240,56.618,-50.631,-179.627,6.287,149.029
C04384=1155.236,56.867,-50.648,-179.624,6.288,149.028
C04385=1155.230,57.117,-50.663,-179.622,6.289,149.028
C04386=1155.225,57.366,-50.679,-179.619,6.290,149.027
C04387=1155.220,57.615,-50.695,-179.617,6.291,149.027
C04388=1155.215,57.865,-50.711,-179.614,6.293,149.026
C04389=1155.210,58.114,-50.728,-179.611,6.293,149.026
C04390=1155.205,58.364,-50.743,-179.609,6.295,149.025
C04391=1155.201,58.613,-50.760,-179.606,6.295,149.025
C04392=1155.195,58.863,-50.776,-179.603,6.297,149.024
C04393=1155.191,59.112,-50.792,-179.601,6.298,149.024
C04394=1155.185,59.362,-50.808,-179.598,6.298,149.023
C04395=1155.181,59.611,-50.825,-179.596,6.300,149.023
C04396=1155.175,59.860,-50.840,-179.593,6.301,149.022
C04397=1155.170,60.109,-50.856,-179.590,6.302,149.022
C04398=1155.166,60.359,-50.872,-179.588,6.303,149.021
C04399=1155.160,60.608,-50.889,-179.585,6.304,149.020
C04400=1155.155,60.858,-50.905,-179.583,6.305,149.020
C04401=1155.150,61.107,-50.922,-179.580,6.307,149.019
C04402=1155.145,61.357,-50.937,-179.577,6.307,149.019
C04403=1155.140,61.606,-50.954,-179.575,6.309,149.018
C04404=1155.136,61.856,-50.970,-179.571,6.310,149.018
C04405=1155.130,62.105,-50.986,-179.569,6.311,149.017
C04406=1155.126,62.355,-51.003,-179.566,6.313,149.017
C04407=1155.120,62.604,-51.018,-179.564,6.313,149.016
C04408=1155.116,62.853,-51.035,-179.561,6.315,149.016
C04409=1155.111,63.103,-51.052,-179.558,6.316,149.015
C04410=1155.105,63.353,-51.068,-179.556,6.317,149.015
C04411=1155.101,63.602,-51.084,-179.553,6.318,149.014
C04412=1155.096,63.851,-51.101,-179.550,6.319,149.014
C04413=1155.091,64.101,-51.117,-179.548,6.320,149.013
C04414=1155.086,64.350,-51.133,-179.545,6.322,149.013
C04415=1155.081,64.599,-51.150,-179.543,6.322,149.012
C04416=1155.075,64.849,-51.166,-179.540,6.324,149.011
C04417=1155.071,65.098,-51.183,-179.537,6.325,149.011
C04418=1155.066,65.348,-51.199,-179.535,6.326,149.011
C04419=1155.061,65.597,-51.216,-179.532,6.327,149.010
C04420=1155.056,65.847,-51.231,-179.529,6.328,149.009
C04421=1155.051,66.096,-51.248,-179.527,6.329,149.009
C04422=1155.046,66.345,-51.265,-179.524,6.331,149.008
C04423=1155.041,66.594,-51.281,-179.521,6.332,149.008
C04424=1155.036,66.844,-51.297,-179.519,6.333,149.007
C04425=1155.032,67.094,-51.314,-179.516,6.334,149.007
C04426=1155.026,67.343,-51.331,-179.514,6.335,149.006
C04427=1155.021,67.592,-51.348,-179.510,6.337,149.006
C04428=1155.016,67.841,-51.364,-179.508,6.337,149.005
C04429=1155.012,68.091,-51.381,-179.505,6.339,149.005
C04430=1155.006,68.341,-51.397,-179.503,6.340,149.004
C04431=1155.001,68.590,-51.413,-179.500,6.341,149.004
C04432=1154.997,68.839,-51.430,-179.497,6.343,149.003
C04433=1154.992,69.089,-51.447,-179.495,6.343,149.003
C04434=1154.987,69.338,-51.464,-179.492,6.345,149.002
C04435=1154.982,69.587,-51.480,-179.489,6.346,149.002
C04436=1154.978,69.837,-51.497,-179.487,6.347,149.001
C04437=1154.972,70.086,-51.514,-179.485,6.348,149.001
C04438=1154.967,70.335,-51.531,-179.481,6.349,149.000
C04439=1154.962,70.586,-51.546,-179.479,6.350,149.000
C04440=1154.957,70.835,-51.563,-179.476,6.352,148.999
C04441=1154.952,71.084,-51.580,-179.473,6.353,148.999
C04442=1154.948,71.334,-51.597,-179.471,6.354,148.998
C04443=1154.942,71.583,-51.614,-179.468,6.355,148.997
C04444=1154.937,71.832,-51.630,-179.466,6.356,148.997
C04445=1154.932,72.082,-51.648,-179.463,6.358,148.997
C04446=1154.927,72.331,-51.664,-179.460,6.359,148.996
C04447=1154.923,72.580,-51.681,-179.458,6.360,148.996
C04448=1154.917,72.830,-51.698,-179.455,6.362,148.995
C04449=1154.912,73.079,-51.714,-179.452,6.362,148.994
C04450=1154.907,73.329,-51.731,-179.449,6.364,148.994
C04451=1154.903,73.578,-51.748,-179.447,6.365,148.993
C04452=1154.898,73.828,-51.765,-179.444,6.366,148.993
C04453=1154.893,74.076,-51.782,-179.441,6.368,148.992
C04454=1154.888,74.326,-51.799,-179.439,6.368,148.992
C04455=1154.883,74.575,-51.816,-179.436,6.370,148.991
C04456=1154.878,74.824,-51.833,-179.434,6.371,148.991
C04457=1154.873,75.074,-51.850,-179.431,6.372,148.990
C04458=1154.868,75.323,-51.866,-179.428,6.374,148.990
C04459=1154.864,75.573,-51.883,-179.426,6.375,148.989
C04460=1154.858,75.822,-51.900,-179.423,6.376,148.989
C04461=1154.853,76.071,-51.917,-179.420,6.377,148.988
C04462=1154.848,76.321,-51.935,-179.418,6.379,148.988
C04463=1154.844,76.570,-51.951,-179.414,6.380,148.987
C04464=1154.839,76.820,-51.969,-179.412,6.381,148.987
C04465=1154.834,77.069,-51.985,-179.410,6.382,148.986
C04466=1154.828,77.318,-52.002,-179.406,6.384,148.986
C04467=1154.824,77.567,-52.020,-179.404,6.385,148.985
C04468=1154.819,77.817,-52.037,-179.401,6.386,148.985
C04469=1154.813,78.066,-52.054,-179.399,6.387,148.984
C04470=1154.809,78.316,-52.070,-179.396,6.389,148.984
C04471=1154.804,78.566,-52.088,-179.393,6.390,148.983
C04472=1154.799,78.814,-52.105,-179.391,6.391,148.983
C04473=1154.794,79.064,-52.122,-179.388,6.392,148.982
C04474=1154.790,79.314,-52.139,-179.385,6.394,148.982
C04475=1154.784,79.582,-52.157,-179.383,6.395,148.981
C04476=1154.779,79.850,-52.177,-179.380,6.396,148.981
C04477=1154.773,80.118,-52.194,-179.377,6.398,148.980
C04478=1154.768,80.387,-52.213,-179.374,6.399,148.980
C04479=1154.763,80.637,-52.230,-179.371,6.401,148.979
C04480=1154.759,80.885,-52.248,-179.369,6.401,148.979
C04481=1154.753,81.135,-52.265,-179.366,6.403,148.978
C04482=1154.748,81.385,-52.282,-179.363,6.404,148.978
C04483=1154.743,81.633,-52.299,-179.360,6.405,148.977
C04484=1154.738,81.883,-52.317,-179.358,6.407,148.977
C04485=1154.734,82.132,-52.334,-179.355,6.407,148.976
C04486=1154.729,82.382,-52.351,-179.352,6.409,148.976
C04487=1154.724,82.631,-52.369,-179.350,6.411,148.975
C04488=1154.719,82.880,-52.386,-179.347,6.411,148.975
C04489=1154.714,83.130,-52.403,-179.344,6.413,148.974
C04490=1154.709,83.379,-52.421,-179.342,6.415,148.974
C04491=1154.703,83.628,-52.438,-179.339,6.415,148.973
C04492=1154.699,83.877,-52.455,-179.336,6.417,148.973
C04493=1154.694,84.127,-52.473,-179.333,6.419,148.972
C04494=1154.689,84.376,-52.491,-179.331,6.419,148.972
C04495=1154.685,84.626,-52.507,-179.328,6.421,148.971
C04496=1154.680,84.875,-52.525,-179.325,6.422,148.971
C04497=1154.674,85.125,-52.543,-179.323,6.423,148.970
C04498=1154.670,85.374,-52.561,-179.320,6.425,148.970
C04499=1154.665,85.623,-52.577,-179.317,6.426,148.969
C04500=1154.660,85.873,-52.595,-179.315,6.427,148.969
C04501=1154.655,86.122,-52.612,-179.312,6.429,148.968
C04502=1154.650,86.372,-52.630,-179.309,6.430,148.968
C04503=1154.646,86.621,-52.647,-179.307,6.431,148.967
C04504=1154.641,86.870,-52.665,-179.304,6.432,148.967
C04505=1154.636,87.119,-52.683,-179.301,6.434,148.966
C04506=1154.630,87.368,-52.700,-179.299,6.435,148.966
C04507=1154.625,87.618,-52.718,-179.296,6.437,148.965
C04508=1154.621,87.867,-52.735,-179.293,6.438,148.965
C04509=1154.616,88.116,-52.753,-179.290,6.440,148.964
C04510=1154.611,88.365,-52.771,-179.288,6.441,148.964
C04511=1154.605,88.615,-52.788,-179.285,6.442,148.963
C04512=1154.601,88.864,-52.806,-179.282,6.444,148.963
C04513=1154.596,89.114,-52.824,-179.280,6.444,148.962
C04514=1154.591,89.363,-52.840,-179.277,6.446,148.962
C04515=1154.586,89.612,-52.858,-179.274,6.447,148.961
C04516=1154.581,89.861,-52.876,-179.272,6.448,148.961
C04517=1154.576,90.111,-52.894,-179.269,6.450,148.961
C04518=1154.571,90.360,-52.912,-179.266,6.451,148.960
C04519=1154.566,90.610,-52.930,-179.263,6.453,148.959
C04520=1154.562,90.859,-52.948,-179.261,6.454,148.959
C04521=1154.557,91.109,-52.966,-179.258,6.456,148.959
C04522=1154.553,91.358,-52.983,-179.255,6.457,148.958
C04523=1154.548,91.607,-53.001,-179.253,6.458,148.958
C04524=1154.543,91.856,-53.019,-179.250,6.459,148.957
C04525=1154.538,92.106,-53.037,-179.247,6.461,148.956
C04526=1154.533,92.355,-53.054,-179.244,6.462,148.956
C04527=1154.528,92.605,-53.072,-179.242,6.463,148.956
C04528=1154.523,92.854,-53.090,-179.239,6.465,148.955
C04529=1154.518,93.103,-53.108,-179.236,6.466,148.955
C04530=1154.513,93.352,-53.126,-179.234,6.468,148.954
C04531=1154.508,93.601,-53.144,-179.231,6.469,148.954
C04532=1154.503,93.850,-53.162,-179.229,6.471,148.953
C04533=1154.498,94.100,-53.179,-179.225,6.472,148.953
C04534=1154.493,94.349,-53.197,-179.223,6.473,148.952
C04535=1154.489,94.599,-53.215,-179.221,6.475,148.952
C04536=1154.484,94.849,-53.233,-179.217,6.476,148.951
C04537=1154.479,95.098,-53.251,-179.215,6.478,148.951
C04538=1154.474,95.347,-53.269,-179.213,6.478,148.950
C04539=1154.469,95.596,-53.287,-179.210,6.480,148.950
C04540=1154.464,95.845,-53.305,-179.207,6.481,148.949
C04541=1154.459,96.094,-53.323,-179.204,6.483,148.949
C04542=1154.454,96.344,-53.341,-179.202,6.484,148.948
C04543=1154.450,96.593,-53.360,-179.199,6.486,148.948
C04544=1154.445,96.843,-53.378,-179.196,6.487,148.947
C04545=1154.440,97.092,-53.396,-179.193,6.489,148.947
C04546=1154.435,97.341,-53.413,-179.191,6.490,148.947
C04547=1154.430,97.590,-53.432,-179.188,6.491,148.946
C04548=1154.425,97.840,-53.450,-179.185,6.493,148.946
C04549=1154.420,98.089,-53.468,-179.182,6.494,148.945
C04550=1154.416,98.339,-53.486,-179.179,6.496,148.945
C04551=1154.411,98.588,-53.504,-179.177,6.497,148.944
C04552=1154.406,98.837,-53.522,-179.174,6.498,148.944
C04553=1154.401,99.086,-53.540,-179.171,6.500,148.943
C04554=1154.396,99.335,-53.558,-179.169,6.502,148.943
C04555=1154.391,99.585,-53.578,-179.167,6.502,148.942
C04556=1154.386,99.834,-53.596,-179.164,6.504,148.942
C04557=1154.381,100.083,-53.614,-179.161,6.505,148.941
C04558=1154.376,100.332,-53.632,-179.158,6.507,148.941
C04559=1154.372,100.582,-53.650,-179.155,6.509,148.940
C04560=1154.367,100.832,-53.668,-179.153,6.510,148.940
C04561=1154.362,101.081,-53.687,-179.150,6.511,148.939
C04562=1154.357,101.330,-53.705,-179.147,6.513,148.939
C04563=1154.352,101.579,-53.723,-179.144,6.514,148.939
C04564=1154.348,101.829,-53.742,-179.142,6.515,148.938
C04565=1154.343,102.078,-53.760,-179.139,6.517,148.938
C04566=1154.337,102.327,-53.778,-179.136,6.518,148.937
C04567=1154.333,102.576,-53.797,-179.134,6.520,148.937
C04568=1154.328,102.826,-53.815,-179.131,6.522,148.936
C04569=1154.323,103.075,-53.833,-179.129,6.523,148.936
C04570=1154.318,103.324,-53.852,-179.125,6.524,148.935
C04571=1154.313,103.573,-53.871,-179.123,6.526,148.935
C04572=1154.309,103.823,-53.889,-179.120,6.527,148.934
C04573=1154.304,104.072,-53.907,-179.117,6.529,148.934
C04574=1154.299,104.321,-53.926,-179.115,6.530,148.933
C04575=1154.294,104.570,-53.944,-179.112,6.531,148.933
C04576=1154.289,104.820,-53.963,-179.109,6.533,148.933
C04577=1154.284,105.069,-53.982,-179.107,6.535,148.932
C04578=1154.279,105.318,-54.000,-179.104,6.536,148.932
C04579=1154.275,105.587,-54.020,-179.101,6.538,148.931
C04580=1154.269,105.855,-54.040,-179.098,6.539,148.931
C04581=1154.264,106.123,-54.060,-179.095,6.541,148.930
C04582=1154.258,106.392,-54.080,-179.092,6.542,148.930
C04583=1154.254,106.641,-54.099,-179.089,6.544,148.929
C04584=1154.248,106.890,-54.117,-179.086,6.546,148.929
C04585=1154.244,107.140,-54.135,-179.084,6.547,148.928
C04586=1154.240,107.389,-54.154,-179.081,6.548,148.928
C04587=1154.234,107.638,-54.173,-179.078,6.550,148.927
C04588=1154.229,107.887,-54.192,-179.076,6.551,148.927
C04589=1154.225,108.137,-54.210,-179.073,6.553,148.927
C04590=1154.220,108.386,-54.229,-179.070,6.555,148.926
C04591=1154.215,108.635,-54.247,-179.068,6.555,148.926
C04592=1154.210,108.884,-54.267,-179.065,6.557,148.925
C04593=1154.205,109.134,-54.285,-179.062,6.559,148.925
C04594=1154.200,109.382,-54.304,-179.059,6.560,148.924
C04595=1154.195,109.632,-54.323,-179.057,6.562,148.924
C04596=1154.191,109.881,-54.341,-179.054,6.564,148.923
C04597=1154.186,110.131,-54.360,-179.051,6.564,148.923
C04598=1154.181,110.380,-54.379,-179.049,6.566,148.922
C04599=1154.176,110.628,-54.398,-179.046,6.568,148.922
C04600=1154.171,110.878,-54.417,-179.043,6.570,148.922
C04601=1154.166,111.127,-54.436,-179.041,6.571,148.921
C04602=1154.162,111.377,-54.454,-179.037,6.573,148.921
C04603=1154.157,111.626,-54.474,-179.035,6.574,148.920
C04604=1154.152,111.875,-54.493,-179.032,6.575,148.920
C04605=1154.147,112.125,-54.511,-179.030,6.577,148.919
C04606=1154.142,112.373,-54.530,-179.027,6.579,148.919
C04607=1154.137,112.623,-54.549,-179.024,6.580,148.919
C04608=1154.133,112.872,-54.567,-179.021,6.582,148.918
C04609=1154.128,113.122,-54.587,-179.018,6.583,148.917
C04610=1154.123,113.370,-54.606,-179.016,6.585,148.917
C04611=1154.118,113.620,-54.625,-179.013,6.587,148.917
C04612=1154.113,113.869,-54.644,-179.011,6.588,148.916
C04613=1154.109,114.118,-54.663,-179.008,6.589,148.916
C04614=1154.103,114.367,-54.682,-179.005,6.591,148.915
C04615=1154.099,114.616,-54.700,-179.002,6.592,148.915
C04616=1154.094,114.866,-54.720,-178.999,6.594,148.914
C04617=1154.088,115.115,-54.739,-178.997,6.596,148.914
C04618=1154.084,115.364,-54.758,-178.994,6.597,148.914
C04619=1154.079,115.614,-54.777,-178.991,6.599,148.913
C04620=1154.075,115.863,-54.796,-178.988,6.601,148.913
C04621=1154.069,116.112,-54.815,-178.986,6.601,148.912
C04622=1154.065,116.361,-54.835,-178.983,6.603,148.912
C04623=1154.060,116.610,-54.854,-178.980,6.605,148.911
C04624=1154.055,116.859,-54.873,-178.978,6.607,148.911
C04625=1154.050,117.110,-54.892,-178.975,6.608,148.911
C04626=1154.046,117.358,-54.911,-178.972,6.610,148.910
C04627=1154.041,117.608,-54.931,-178.969,6.611,148.910
C04628=1154.036,117.857,-54.950,-178.966,6.613,148.909
C04629=1154.032,118.106,-54.969,-178.964,6.615,148.909
C04630=1154.026,118.355,-54.988,-178.961,6.616,148.908
C04631=1154.022,118.604,-55.008,-178.958,6.618,148.908
C04632=1154.017,118.853,-55.027,-178.956,6.619,148.908
C04633=1154.012,119.102,-55.046,-178.953,6.621,148.907
C04634=1154.007,119.351,-55.066,-178.951,6.622,148.907
C04635=1154.002,119.601,-55.085,-178.947,6.624,148.906
C04636=1153.998,119.850,-55.104,-178.945,6.625,148.906
C04637=1153.993,120.099,-55.124,-178.942,6.627,148.905
C04638=1153.988,120.349,-55.143,-178.939,6.629,148.905
C04639=1153.983,120.597,-55.163,-178.937,6.631,148.904
C04640=1153.979,120.847,-55.182,-178.934,6.632,148.904
C04641=1153.974,121.096,-55.201,-178.931,6.634,148.904
C04642=1153.969,121.345,-55.221,-178.928,6.636,148.903
C04643=1153.964,121.595,-55.240,-178.925,6.637,148.903
C04644=1153.959,121.844,-55.259,-178.923,6.639,148.902
C04645=1153.955,122.093,-55.279,-178.920,6.640,148.902
C04646=1153.950,122.342,-55.298,-178.918,6.641,148.901
C04647=1153.944,122.591,-55.317,-178.915,6.643,148.901
C04648=1153.940,122.841,-55.337,-178.912,6.645,148.901
C04649=1153.935,123.090,-55.357,-178.910,6.646,148.900
C04650=1153.930,123.339,-55.376,-178.907,6.648,148.900
C04651=1153.926,123.588,-55.396,-178.904,6.650,148.899
C04652=1153.921,123.838,-55.416,-178.901,6.651,148.899
C04653=1153.916,124.086,-55.435,-178.898,6.653,148.898
C04654=1153.911,124.336,-55.454,-178.895,6.655,148.898
C04655=1153.906,124.586,-55.474,-178.893,6.656,148.898
C04656=1153.901,124.834,-55.493,-178.890,6.658,148.897
C04657=1153.897,125.083,-55.514,-178.887,6.660,148.897
C04658=1153.893,125.333,-55.533,-178.885,6.662,148.896
C04659=1153.887,125.581,-55.552,-178.882,6.663,148.896
C04660=1153.882,125.831,-55.572,-178.879,6.665,148.896
C04661=1153.878,126.080,-55.592,-178.876,6.667,148.895
C04662=1153.873,126.329,-55.611,-178.874,6.668,148.895
C04663=1153.868,126.578,-55.631,-178.871,6.670,148.894
C04664=1153.863,126.828,-55.651,-178.868,6.671,148.894
C04665=1153.859,127.077,-55.671,-178.865,6.673,148.893
C04666=1153.853,127.326,-55.690,-178.862,6.675,148.893
C04667=1153.849,127.575,-55.710,-178.860,6.677,148.893
C04668=1153.844,127.824,-55.730,-178.857,6.678,148.892
C04669=1153.839,128.074,-55.750,-178.854,6.680,148.892
C04670=1153.834,128.323,-55.769,-178.852,6.682,148.891
C04671=1153.830,128.572,-55.790,-178.849,6.683,148.891
C04672=1153.825,128.821,-55.809,-178.846,6.685,148.891
C04673=1153.820,129.070,-55.829,-178.843,6.687,148.890
C04674=1153.815,129.319,-55.849,-178.841,6.689,148.890
C04675=1153.810,129.569,-55.869,-178.838,6.690,148.889
C04676=1153.806,129.818,-55.889,-178.835,6.692,148.889
C04677=1153.801,130.067,-55.909,-178.832,6.693,148.888
C04678=1153.796,130.315,-55.929,-178.829,6.695,148.888
C04679=1153.791,130.565,-55.948,-178.827,6.697,148.888
C04680=1153.787,130.815,-55.968,-178.824,6.698,148.887
C04681=1153.782,131.063,-55.988,-178.821,6.700,148.887
C04682=1153.777,131.312,-56.008,-178.819,6.702,148.886
C04683=1153.772,131.581,-56.030,-178.816,6.704,148.886
C04684=1153.767,131.849,-56.051,-178.813,6.705,148.886
C04685=1153.761,132.118,-56.073,-178.810,6.707,148.885
C04686=1153.756,132.386,-56.095,-178.807,6.709,148.885
C04687=1153.752,132.636,-56.114,-178.804,6.711,148.884
C04688=1153.747,132.885,-56.135,-178.801,6.713,148.884
C04689=1153.742,133.135,-56.155,-178.798,6.714,148.884
C04690=1153.737,133.384,-56.175,-178.796,6.716,148.883
C04691=1153.733,133.633,-56.196,-178.793,6.718,148.883
C04692=1153.728,133.881,-56.215,-178.790,6.719,148.882
C04693=1153.723,134.130,-56.235,-178.788,6.721,148.882
C04694=1153.718,134.380,-56.255,-178.785,6.723,148.882
C04695=1153.713,134.629,-56.276,-178.782,6.725,148.881
C04696=1153.709,134.878,-56.296,-178.779,6.726,148.881
C04697=1153.704,135.128,-56.316,-178.777,6.728,148.880
C04698=1153.700,135.377,-56.336,-178.774,6.730,148.880
C04699=1153.695,135.625,-56.356,-178.771,6.732,148.880
C04700=1153.689,135.875,-56.377,-178.769,6.733,148.879
C04701=1153.685,136.124,-56.397,-178.766,6.735,148.879
C04702=1153.680,136.373,-56.417,-178.763,6.737,148.878
C04703=1153.675,136.622,-56.437,-178.760,6.738,148.878
C04704=1153.670,136.872,-56.458,-178.758,6.740,148.878
C04705=1153.666,137.121,-56.478,-178.755,6.742,148.877
C04706=1153.661,137.369,-56.499,-178.752,6.744,148.877
C04707=1153.657,137.619,-56.518,-178.750,6.745,148.876
C04708=1153.651,137.868,-56.539,-178.747,6.747,148.876
C04709=1153.647,138.117,-56.560,-178.744,6.749,148.876
C04710=1153.643,138.366,-56.580,-178.741,6.751,148.875
C04711=1153.637,138.615,-56.601,-178.738,6.753,148.875
C04712=1153.632,138.864,-56.620,-178.736,6.755,148.875
C04713=1153.628,139.113,-56.641,-178.733,6.756,148.874
C04714=1153.622,139.363,-56.662,-178.730,6.758,148.874
C04715=1153.618,139.611,-56.682,-178.727,6.760,148.873
C04716=1153.614,139.860,-56.703,-178.725,6.762,148.873
C04717=1153.608,140.110,-56.723,-178.722,6.763,148.873
C04718=1153.604,140.359,-56.744,-178.719,6.765,148.872
C04719=1153.600,140.608,-56.764,-178.717,6.767,148.872
C04720=1153.594,140.857,-56.784,-178.714,6.768,148.871
C04721=1153.590,141.106,-56.805,-178.711,6.770,148.871
C04722=1153.585,141.355,-56.825,-178.708,6.772,148.871
C04723=1153.580,141.605,-56.846,-178.705,6.774,148.870
C04724=1153.576,141.854,-56.867,-178.702,6.776,148.870
C04725=1153.570,142.103,-56.888,-178.700,6.778,148.869
C04726=1153.566,142.352,-56.908,-178.697,6.780,148.869
C04727=1153.562,142.601,-56.928,-178.694,6.781,148.869
C04728=1153.556,142.850,-56.949,-178.692,6.783,148.868
C04729=1153.552,143.099,-56.970,-178.689,6.785,148.868
C04730=1153.547,143.348,-56.991,-178.686,6.786,148.868
C04731=1153.542,143.597,-57.011,-178.683,6.788,148.867
C04732=1153.538,143.847,-57.032,-178.681,6.790,148.867
C04733=1153.533,144.096,-57.053,-178.678,6.792,148.866
C04734=1153.528,144.345,-57.074,-178.675,6.794,148.866
C04735=1153.524,144.594,-57.094,-178.672,6.796,148.866
C04736=1153.519,144.843,-57.116,-178.669,6.798,148.865
C04737=1153.514,145.092,-57.136,-178.667,6.799,148.865
C04738=1153.509,145.341,-57.157,-178.664,6.801,148.864
C04739=1153.505,145.590,-57.177,-178.661,6.803,148.864
C04740=1153.500,145.839,-57.198,-178.658,6.804,148.864
C04741=1153.495,146.088,-57.219,-178.656,6.806,148.863
C04742=1153.490,146.338,-57.240,-178.652,6.809,148.863
C04743=1153.486,146.586,-57.261,-178.650,6.810,148.863
C04744=1153.481,146.835,-57.282,-178.647,6.812,148.862
C04745=1153.477,147.085,-57.302,-178.644,6.814,148.862
C04746=1153.472,147.334,-57.323,-178.642,6.816,148.862
C04747=1153.466,147.583,-57.344,-178.639,6.818,148.861
C04748=1153.462,147.832,-57.365,-178.637,6.819,148.861
C04749=1153.457,148.081,-57.386,-178.634,6.821,148.860
C04750=1153.453,148.330,-57.407,-178.631,6.824,148.860
C04751=1153.448,148.579,-57.428,-178.628,6.825,148.860
C04752=1153.443,148.828,-57.449,-178.625,6.827,148.859
C04753=1153.439,149.077,-57.470,-178.623,6.829,148.859
C04754=1153.434,149.327,-57.491,-178.620,6.831,148.859
C04755=1153.430,149.575,-57.512,-178.617,6.832,148.858
C04756=1153.424,149.824,-57.533,-178.615,6.834,148.858
C04757=1153.419,150.074,-57.554,-178.611,6.837,148.857
C04758=1153.415,150.322,-57.575,-178.609,6.838,148.857
C04759=1153.410,150.572,-57.597,-178.606,6.840,148.857
C04760=1153.405,150.821,-57.618,-178.603,6.842,148.856
C04761=1153.400,151.070,-57.639,-178.601,6.844,148.856
C04762=1153.396,151.319,-57.660,-178.598,6.846,148.856
C04763=1153.391,151.568,-57.681,-178.595,6.847,148.855
C04764=1153.387,151.817,-57.703,-178.592,6.850,148.855
C04765=1153.382,152.066,-57.723,-178.589,6.852,148.855
C04766=1153.377,152.315,-57.745,-178.587,6.853,148.854
C04767=1153.372,152.564,-57.766,-178.584,6.855,148.854
C04768=1153.367,152.813,-57.787,-178.581,6.857,148.854
C04769=1153.363,153.062,-57.808,-178.579,6.858,148.853
C04770=1153.358,153.312,-57.829,-178.575,6.861,148.853
C04771=1153.353,153.560,-57.851,-178.573,6.863,148.852
C04772=1153.348,153.810,-57.872,-178.570,6.865,148.852
C04773=1153.345,154.059,-57.893,-178.568,6.867,148.852
C04774=1153.340,154.307,-57.915,-178.565,6.868,148.851
C04775=1153.335,154.556,-57.936,-178.562,6.871,148.851
C04776=1153.330,154.805,-57.958,-178.559,6.873,148.851
C04777=1153.325,155.055,-57.979,-178.556,6.874,148.850
C04778=1153.320,155.304,-58.001,-178.554,6.876,148.850
C04779=1153.316,155.553,-58.021,-178.551,6.878,148.850
C04780=1153.311,155.801,-58.043,-178.548,6.879,148.849
C04781=1153.307,156.051,-58.065,-178.545,6.882,148.849
C04782=1153.302,156.300,-58.086,-178.543,6.884,148.849
C04783=1153.297,156.549,-58.107,-178.540,6.886,148.848
C04784=1153.292,156.799,-58.129,-178.537,6.888,148.848
C04785=1153.287,157.047,-58.150,-178.535,6.889,148.848
C04786=1153.283,157.295,-58.171,-178.531,6.892,148.847
C04787=1153.278,157.565,-58.195,-178.529,6.894,148.847
C04788=1153.273,157.834,-58.217,-178.525,6.896,148.846
C04789=1153.268,158.103,-58.242,-178.523,6.898,148.846
C04790=1153.263,158.372,-58.264,-178.519,6.900,148.846
C04791=1153.258,158.620,-58.286,-178.517,6.902,148.845
C04792=1153.253,158.870,-58.307,-178.514,6.904,148.845
C04793=1153.249,159.119,-58.329,-178.512,6.906,148.845
C04794=1153.244,159.368,-58.351,-178.509,6.908,148.844
C04795=1153.239,159.617,-58.373,-178.506,6.910,148.844
C04796=1153.234,159.866,-58.394,-178.503,6.912,148.844
C04797=1153.229,160.115,-58.415,-178.500,6.914,148.843
C04798=1153.225,160.364,-58.437,-178.498,6.915,148.843
C04799=1153.220,160.613,-58.459,-178.494,6.918,148.843
C04800=1153.216,160.862,-58.481,-178.492,6.920,148.842
C04801=1153.211,161.111,-58.503,-178.489,6.922,148.842
C04802=1153.206,161.360,-58.524,-178.487,6.924,148.842
C04803=1153.202,161.609,-58.546,-178.484,6.925,148.841
C04804=1153.197,161.858,-58.568,-178.481,6.928,148.841
C04805=1153.193,162.107,-58.590,-178.478,6.930,148.841
C04806=1153.188,162.356,-58.611,-178.476,6.932,148.840
C04807=1153.183,162.605,-58.633,-178.473,6.933,148.840
C04808=1153.179,162.854,-58.655,-178.470,6.936,148.840
C04809=1153.174,163.103,-58.677,-178.467,6.938,148.839
C04810=1153.169,163.352,-58.699,-178.464,6.939,148.839
C04811=1153.165,163.601,-58.720,-178.462,6.941,148.839
C04812=1153.160,163.850,-58.743,-178.459,6.944,148.838
C04813=1153.155,164.099,-58.765,-178.456,6.946,148.838
C04814=1153.150,164.348,-58.787,-178.454,6.947,148.838
C04815=1153.146,164.597,-58.809,-178.451,6.949,148.837
C04816=1153.141,164.846,-58.831,-178.448,6.952,148.837
C04817=1153.136,165.095,-58.852,-178.445,6.954,148.837
C04818=1153.132,165.343,-58.874,-178.443,6.956,148.836
C04819=1153.127,165.593,-58.896,-178.439,6.958,148.836
C04820=1153.122,165.841,-58.918,-178.437,6.960,148.836
C04821=1153.117,166.091,-58.940,-178.434,6.962,148.835
C04822=1153.113,166.340,-58.962,-178.432,6.964,148.835
C04823=1153.108,166.589,-58.984,-178.428,6.966,148.835
C04824=1153.103,166.838,-59.006,-178.426,6.968,148.834
C04825=1153.099,167.087,-59.028,-178.423,6.970,148.834
C04826=1153.094,167.335,-59.051,-178.420,6.971,148.834
C04827=1153.090,167.585,-59.073,-178.418,6.974,148.834
C04828=1153.085,167.834,-59.095,-178.415,6.976,148.833
C04829=1153.080,168.083,-59.117,-178.412,6.978,148.833
C04830=1153.076,168.332,-59.139,-178.409,6.980,148.833
C04831=1153.071,168.581,-59.161,-178.406,6.982,148.832
C04832=1153.067,168.830,-59.184,-178.404,6.984,148.832
C04833=1153.062,169.078,-59.205,-178.401,6.986,148.832
C04834=1153.057,169.328,-59.228,-178.398,6.988,148.831
C04835=1153.052,169.577,-59.250,-178.395,6.990,148.831
C04836=1153.048,169.825,-59.272,-178.393,6.992,148.831
C04837=1153.043,170.074,-59.294,-178.390,6.995,148.830
C04838=1153.038,170.324,-59.317,-178.387,6.997,148.830
C04839=1153.034,170.573,-59.339,-178.384,6.998,148.830
C04840=1153.029,170.821,-59.361,-178.381,7.001,148.829
C04841=1153.024,171.071,-59.384,-178.379,7.003,148.829
C04842=1153.019,171.319,-59.405,-178.376,7.005,148.829
C04843=1153.015,171.568,-59.428,-178.373,7.006,148.828
C04844=1153.010,171.818,-59.451,-178.370,7.009,148.828
C04845=1153.005,172.066,-59.473,-178.368,7.011,148.828
C04846=1153.002,172.315,-59.495,-178.365,7.013,148.828
C04847=1152.996,172.564,-59.518,-178.362,7.015,148.827
C04848=1152.992,172.813,-59.540,-178.359,7.017,148.827
C04849=1152.987,173.062,-59.563,-178.357,7.019,148.827
C04850=1152.982,173.311,-59.585,-178.354,7.022,148.826
C04851=1152.978,173.560,-59.607,-178.351,7.024,148.826
C04852=1152.973,173.809,-59.630,-178.348,7.025,148.826
C04853=1152.969,174.057,-59.653,-178.346,7.028,148.825
C04854=1152.964,174.307,-59.675,-178.343,7.030,148.825
C04855=1152.960,174.556,-59.698,-178.340,7.032,148.825
C04856=1152.955,174.804,-59.720,-178.337,7.034,148.824
C04857=1152.950,175.053,-59.743,-178.335,7.036,148.824
C04858=1152.946,175.303,-59.765,-178.332,7.038,148.824
C04859=1152.940,175.551,-59.788,-178.329,7.041,148.824
C04860=1152.936,175.800,-59.810,-178.327,7.043,148.823
C04861=1152.931,176.050,-59.833,-178.324,7.044,148.823
C04862=1152.927,176.298,-59.855,-178.321,7.047,148.823
C04863=1152.922,176.547,-59.878,-178.318,7.049,148.822
C04864=1152.918,176.796,-59.901,-178.316,7.051,148.822
C04865=1152.912,177.045,-59.923,-178.312,7.053,148.822
C04866=1152.908,177.294,-59.946,-178.310,7.055,148.821
C04867=1152.903,177.543,-59.969,-178.307,7.058,148.821
C04868=1152.899,177.792,-59.992,-178.304,7.060,148.821
C04869=1152.894,178.040,-60.015,-178.302,7.061,148.821
C04870=1152.890,178.290,-60.037,-178.298,7.064,148.820
C04871=1152.885,178.539,-60.060,-178.296,7.066,148.820
C04872=1152.880,178.788,-60.083,-178.293,7.068,148.820
C04873=1152.876,179.036,-60.105,-178.290,7.070,148.819
C04874=1152.871,179.285,-60.128,-178.288,7.073,148.819
C04875=1152.867,179.534,-60.151,-178.285,7.074,148.819
C04876=1152.862,179.783,-60.175,-178.282,7.077,148.819
C04877=1152.857,180.032,-60.196,-178.280,7.079,148.818
C04878=1152.853,180.281,-60.220,-178.276,7.081,148.818
C04879=1152.848,180.530,-60.243,-178.274,7.083,148.818
C04880=1152.844,180.779,-60.266,-178.271,7.085,148.818
C04881=1152.839,181.028,-60.288,-178.268,7.088,148.817
C04882=1152.834,181.277,-60.311,-178.266,7.090,148.817
C04883=1152.830,181.525,-60.334,-178.262,7.092,148.817
C04884=1152.825,181.774,-60.358,-178.260,7.094,148.816
C04885=1152.820,182.023,-60.381,-178.257,7.096,148.816
C04886=1152.816,182.272,-60.404,-178.254,7.099,148.816
C04887=1152.811,182.522,-60.426,-178.252,7.101,148.816
C04888=1152.806,182.770,-60.449,-178.249,7.102,148.815
C04889=1152.802,183.019,-60.472,-178.246,7.105,148.815
C04890=1152.797,183.268,-60.495,-178.244,7.107,148.815
C04891=1152.792,183.538,-60.520,-178.240,7.110,148.814
C04892=1152.787,183.807,-60.545,-178.237,7.112,148.814
C04893=1152.782,184.076,-60.571,-178.234,7.114,148.814
C04894=1152.777,184.346,-60.596,-178.232,7.117,148.814
C04895=1152.772,184.595,-60.619,-178.229,7.119,148.813
C04896=1152.768,184.844,-60.642,-178.226,7.121,148.813
C04897=1152.764,185.093,-60.665,-178.223,7.123,148.813
C04898=1152.759,185.342,-60.688,-178.220,7.126,148.812
C04899=1152.754,185.591,-60.712,-178.217,7.128,148.812
C04900=1152.750,185.840,-60.735,-178.215,7.130,148.812
C04901=1152.746,186.089,-60.758,-178.212,7.132,148.812
C04902=1152.740,186.337,-60.781,-178.209,7.134,148.811
C04903=1152.736,186.586,-60.804,-178.206,7.137,148.811
C04904=1152.731,186.835,-60.828,-178.204,7.139,148.811
C04905=1152.726,187.084,-60.851,-178.201,7.142,148.811
C04906=1152.722,187.333,-60.874,-178.198,7.143,148.810
C04907=1152.718,187.582,-60.897,-178.195,7.146,148.810
C04908=1152.713,187.831,-60.921,-178.193,7.148,148.810
C04909=1152.709,188.079,-60.945,-178.190,7.150,148.809
C04910=1152.704,188.328,-60.968,-178.187,7.153,148.809
C04911=1152.699,188.577,-60.991,-178.185,7.154,148.809
C04912=1152.694,188.826,-61.015,-178.181,7.157,148.809
C04913=1152.690,189.075,-61.038,-178.179,7.159,148.808
C04914=1152.685,189.324,-61.061,-178.176,7.162,148.808
C04915=1152.681,189.573,-61.085,-178.173,7.163,148.808
C04916=1152.677,189.821,-61.108,-178.170,7.166,148.808
C04917=1152.672,190.070,-61.132,-178.168,7.168,148.807
C04918=1152.667,190.320,-61.155,-178.166,7.170,148.807
C04919=1152.663,190.568,-61.179,-178.162,7.173,148.807
C04920=1152.658,190.817,-61.202,-178.160,7.174,148.806
C04921=1152.653,191.066,-61.226,-178.157,7.177,148.806
C04922=1152.649,191.315,-61.249,-178.154,7.179,148.806
C04923=1152.644,191.563,-61.273,-178.151,7.182,148.806
C04924=1152.640,191.812,-61.297,-178.149,7.184,148.806
C04925=1152.635,192.061,-61.320,-178.146,7.187,148.805
C04926=1152.631,192.310,-61.344,-178.143,7.188,148.805
C04927=1152.626,192.559,-61.367,-178.140,7.191,148.805
C04928=1152.622,192.807,-61.391,-178.138,7.193,148.805
C04929=1152.617,193.056,-61.415,-178.134,7.196,148.804
C04930=1152.612,193.305,-61.438,-178.132,7.198,148.804
C04931=1152.608,193.554,-61.462,-178.129,7.200,148.804
C04932=1152.603,193.803,-61.486,-178.127,7.202,148.804
C04933=1152.598,194.052,-61.510,-178.123,7.205,148.803
C04934=1152.593,194.301,-61.534,-178.121,7.207,148.803
C04935=1152.588,194.550,-61.557,-178.118,7.209,148.803
C04936=1152.584,194.798,-61.581,-178.115,7.211,148.803
C04937=1152.579,195.047,-61.604,-178.113,7.213,148.802
C04938=1152.575,195.295,-61.628,-178.110,7.216,148.802
C04939=1152.570,195.545,-61.652,-178.108,7.218,148.802
C04940=1152.567,195.794,-61.676,-178.104,7.221,148.802
C04941=1152.562,196.043,-61.700,-178.102,7.223,148.801
C04942=1152.557,196.291,-61.724,-178.099,7.225,148.801
C04943=1152.552,196.540,-61.748,-178.096,7.227,148.801
C04944=1152.548,196.789,-61.772,-178.093,7.230,148.801
C04945=1152.543,197.037,-61.796,-178.091,7.232,148.800
C04946=1152.538,197.286,-61.819,-178.088,7.235,148.800
C04947=1152.534,197.535,-61.843,-178.085,7.236,148.800
C04948=1152.529,197.785,-61.868,-178.082,7.239,148.800
C04949=1152.525,198.033,-61.892,-178.079,7.242,148.799
C04950=1152.520,198.282,-61.916,-178.077,7.244,148.799
C04951=1152.516,198.531,-61.939,-178.074,7.247,148.799
C04952=1152.511,198.779,-61.963,-178.071,7.249,148.799
C04953=1152.506,199.028,-61.988,-178.068,7.251,148.799
C04954=1152.502,199.277,-62.011,-178.066,7.253,148.798
C04955=1152.498,199.526,-62.036,-178.063,7.256,148.798
C04956=1152.493,199.774,-62.060,-178.060,7.258,148.798
C04957=1152.488,200.023,-62.084,-178.057,7.261,148.798
C04958=1152.484,200.272,-62.108,-178.055,7.263,148.797
C04959=1152.479,200.520,-62.132,-178.052,7.265,148.797
C04960=1152.475,200.770,-62.156,-178.049,7.267,148.797
C04961=1152.470,201.018,-62.181,-178.046,7.270,148.797
C04962=1152.466,201.267,-62.204,-178.044,7.272,148.797
C04963=1152.461,201.516,-62.228,-178.041,7.275,148.796
C04964=1152.457,201.765,-62.253,-178.039,7.277,148.796
C04965=1152.452,202.014,-62.277,-178.035,7.279,148.796
C04966=1152.448,202.262,-62.301,-178.032,7.282,148.796
C04967=1152.443,202.511,-62.326,-178.030,7.284,148.795
C04968=1152.439,202.760,-62.350,-178.027,7.287,148.795
C04969=1152.434,203.009,-62.374,-178.024,7.289,148.795
C04970=1152.429,203.258,-62.399,-178.022,7.292,148.795
C04971=1152.425,203.506,-62.423,-178.019,7.293,148.794
C04972=1152.421,203.755,-62.447,-178.016,7.296,148.794
C04973=1152.416,204.004,-62.472,-178.013,7.298,148.794
C04974=1152.411,204.252,-62.496,-178.011,7.301,148.794
C04975=1152.406,204.501,-62.521,-178.007,7.304,148.794
C04976=1152.402,204.750,-62.545,-178.005,7.306,148.793
C04977=1152.398,204.999,-62.569,-178.002,7.308,148.793
C04978=1152.393,205.247,-62.594,-178.000,7.310,148.793
C04979=1152.389,205.496,-62.618,-177.996,7.313,148.793
C04980=1152.384,205.745,-62.643,-177.994,7.315,148.793
C04981=1152.380,205.993,-62.667,-177.991,7.318,148.792
C04982=1152.374,206.242,-62.692,-177.988,7.320,148.792
C04983=1152.371,206.491,-62.716,-177.986,7.323,148.792
C04984=1152.366,206.740,-62.741,-177.983,7.325,148.792
C04985=1152.361,206.988,-62.765,-177.980,7.327,148.792
C04986=1152.357,207.238,-62.790,-177.977,7.330,148.791
C04987=1152.352,207.486,-62.814,-177.975,7.332,148.791
C04988=1152.347,207.735,-62.839,-177.972,7.335,148.791
C04989=1152.343,207.984,-62.863,-177.969,7.337,148.791
C04990=1152.338,208.232,-62.888,-177.967,7.340,148.791
C04991=1152.335,208.481,-62.913,-177.963,7.342,148.790
C04992=1152.330,208.730,-62.937,-177.961,7.344,148.790
C04993=1152.324,208.979,-62.962,-177.958,7.347,148.790
C04994=1152.321,209.228,-62.987,-177.955,7.350,148.790
C04995=1152.315,209.498,-63.013,-177.952,7.352,148.789
C04996=1152.311,209.769,-63.040,-177.950,7.354,148.789
C04997=1152.306,210.039,-63.067,-177.946,7.357,148.789
C04998=1152.301,210.310,-63.094,-177.944,7.360,148.789
C04999=1152.296,210.559,-63.119,-177.940,7.362,148.788
C05000=1152.291,210.807,-63.144,-177.938,7.365,148.788
C05001=1152.287,211.056,-63.169,-177.935,7.367,148.788
C05002=1152.282,211.305,-63.193,-177.932,7.370,148.788
C05003=1152.278,211.553,-63.219,-177.930,7.372,148.788
C05004=1152.274,211.802,-63.243,-177.927,7.375,148.788
C05005=1152.269,212.051,-63.268,-177.924,7.378,148.787
C05006=1152.264,212.299,-63.294,-177.921,7.379,148.787
C05007=1152.260,212.548,-63.318,-177.918,7.382,148.787
C05008=1152.255,212.797,-63.343,-177.916,7.384,148.787
C05009=1152.251,213.045,-63.368,-177.913,7.387,148.787
C05010=1152.247,213.294,-63.393,-177.910,7.390,148.786
C05011=1152.242,213.543,-63.418,-177.908,7.392,148.786
C05012=1152.237,213.792,-63.443,-177.905,7.395,148.786
C05013=1152.232,214.041,-63.468,-177.902,7.398,148.786
C05014=1152.229,214.289,-63.493,-177.899,7.399,148.786
C05015=1152.224,214.538,-63.517,-177.896,7.402,148.785
C05016=1152.219,214.787,-63.543,-177.894,7.405,148.785
C05017=1152.214,215.035,-63.568,-177.891,7.407,148.785
C05018=1152.211,215.284,-63.593,-177.888,7.410,148.785
C05019=1152.206,215.533,-63.618,-177.885,7.413,148.785
C05020=1152.201,215.781,-63.643,-177.883,7.415,148.784
C05021=1152.196,216.030,-63.668,-177.880,7.417,148.784
C05022=1152.193,216.279,-63.693,-177.878,7.420,148.784
C05023=1152.188,216.527,-63.718,-177.874,7.422,148.784
C05024=1152.183,216.776,-63.744,-177.872,7.425,148.784
C05025=1152.179,217.024,-63.769,-177.869,7.427,148.784
C05026=1152.174,217.274,-63.794,-177.866,7.430,148.783
C05027=1152.170,217.523,-63.820,-177.863,7.433,148.783
C05028=1152.166,217.771,-63.844,-177.861,7.434,148.783
C05029=1152.161,218.020,-63.870,-177.858,7.437,148.783
C05030=1152.156,218.268,-63.895,-177.855,7.440,148.783
C05031=1152.152,218.517,-63.920,-177.852,7.442,148.782
C05032=1152.147,218.765,-63.945,-177.850,7.445,148.782
C05033=1152.143,219.014,-63.971,-177.847,7.448,148.782
C05034=1152.138,219.264,-63.996,-177.844,7.450,148.782
C05035=1152.134,219.512,-64.022,-177.841,7.453,148.782
C05036=1152.129,219.761,-64.047,-177.839,7.456,148.782
C05037=1152.124,220.009,-64.073,-177.835,7.458,148.781
C05038=1152.121,220.258,-64.097,-177.833,7.460,148.781
C05039=1152.116,220.507,-64.123,-177.830,7.463,148.781
C05040=1152.112,220.755,-64.148,-177.828,7.466,148.781
C05041=1152.107,221.003,-64.174,-177.825,7.468,148.781
C05042=1152.103,221.252,-64.200,-177.822,7.471,148.781
C05043=1152.098,221.501,-64.225,-177.819,7.474,148.781
C05044=1152.094,221.750,-64.250,-177.817,7.475,148.780
C05045=1152.089,221.998,-64.276,-177.814,7.478,148.780
C05046=1152.085,222.247,-64.301,-177.811,7.481,148.780
C05047=1152.081,222.496,-64.327,-177.808,7.484,148.780
C05048=1152.076,222.744,-64.353,-177.806,7.486,148.780
C05049=1152.072,222.992,-64.378,-177.803,7.489,148.780
C05050=1152.067,223.242,-64.403,-177.800,7.491,148.779
C05051=1152.062,223.490,-64.429,-177.797,7.494,148.779
C05052=1152.057,223.739,-64.455,-177.795,7.497,148.779
C05053=1152.053,223.988,-64.481,-177.792,7.499,148.779
C05054=1152.049,224.237,-64.507,-177.789,7.501,148.779
C05055=1152.044,224.485,-64.532,-177.786,7.504,148.779
C05056=1152.040,224.734,-64.558,-177.784,7.507,148.779
C05057=1152.035,224.982,-64.583,-177.781,7.510,148.778
C05058=1152.031,225.230,-64.609,-177.778,7.512,148.778
C05059=1152.026,225.479,-64.635,-177.775,7.515,148.778
C05060=1152.022,225.728,-64.660,-177.773,7.518,148.778
C05061=1152.018,225.977,-64.686,-177.769,7.520,148.778
C05062=1152.012,226.225,-64.712,-177.767,7.522,148.777
C05063=1152.008,226.474,-64.738,-177.764,7.525,148.777
C05064=1152.004,226.722,-64.764,-177.761,7.528,148.777
C05065=1152.000,226.971,-64.790,-177.758,7.531,148.777
C05066=1151.995,227.219,-64.815,-177.756,7.533,148.777
C05067=1151.991,227.468,-64.841,-177.753,7.536,148.777
C05068=1151.986,227.717,-64.868,-177.750,7.539,148.777
C05069=1151.982,227.966,-64.893,-177.747,7.541,148.776
C05070=1151.977,228.214,-64.919,-177.745,7.543,148.776
C05071=1151.973,228.462,-64.945,-177.742,7.546,148.776
C05072=1151.968,228.711,-64.971,-177.739,7.549,148.776
C05073=1151.964,228.960,-64.997,-177.736,7.552,148.776
C05074=1151.960,229.209,-65.023,-177.734,7.554,148.776
C05075=1151.955,229.457,-65.048,-177.731,7.557,148.776
C05076=1151.950,229.706,-65.075,-177.728,7.560,148.776
C05077=1151.946,229.954,-65.101,-177.726,7.563,148.775
C05078=1151.942,230.203,-65.127,-177.723,7.565,148.775
C05079=1151.937,230.452,-65.153,-177.720,7.567,148.775
C05080=1151.932,230.700,-65.179,-177.717,7.570,148.775
C05081=1151.928,230.949,-65.205,-177.715,7.573,148.775
C05082=1151.924,231.197,-65.231,-177.712,7.575,148.775
C05083=1151.919,231.446,-65.258,-177.709,7.578,148.774
C05084=1151.915,231.695,-65.284,-177.706,7.581,148.774
C05085=1151.911,231.943,-65.309,-177.704,7.584,148.774
C05086=1151.906,232.192,-65.337,-177.701,7.587,148.774
C05087=1151.901,232.440,-65.362,-177.698,7.589,148.774
C05088=1151.897,232.688,-65.388,-177.695,7.591,148.774
C05089=1151.892,232.937,-65.415,-177.693,7.594,148.774
C05090=1151.888,233.186,-65.440,-177.690,7.597,148.774
C05091=1151.883,233.435,-65.468,-177.688,7.599,148.774
C05092=1151.879,233.683,-65.493,-177.684,7.602,148.773
C05093=1151.875,233.932,-65.520,-177.682,7.605,148.773
C05094=1151.870,234.181,-65.546,-177.679,7.608,148.773
C05095=1151.866,234.429,-65.573,-177.676,7.611,148.773
C05096=1151.861,234.678,-65.599,-177.674,7.613,148.773
C05097=1151.857,234.926,-65.625,-177.671,7.616,148.773
C05098=1151.852,235.175,-65.651,-177.668,7.618,148.773
C05099=1151.848,235.447,-65.680,-177.665,7.621,148.772
C05100=1151.843,235.718,-65.710,-177.662,7.624,148.772
C05101=1151.838,235.990,-65.738,-177.658,7.628,148.772
C05102=1151.833,236.262,-65.767,-177.656,7.631,148.772
C05103=1151.829,236.511,-65.793,-177.653,7.634,148.772
C05104=1151.824,236.759,-65.820,-177.651,7.636,148.772
C05105=1151.820,237.007,-65.846,-177.648,7.639,148.772
C05106=1151.815,237.256,-65.873,-177.645,7.642,148.772
C05107=1151.812,237.505,-65.899,-177.642,7.644,148.771
C05108=1151.807,237.753,-65.926,-177.639,7.647,148.771
C05109=1151.802,238.002,-65.953,-177.637,7.649,148.771
C05110=1151.798,238.250,-65.979,-177.634,7.652,148.771
C05111=1151.793,238.499,-66.006,-177.631,7.655,148.771
C05112=1151.789,238.748,-66.032,-177.628,7.658,148.771
C05113=1151.784,238.996,-66.059,-177.625,7.661,148.771
C05114=1151.781,239.244,-66.085,-177.622,7.664,148.771
C05115=1151.776,239.493,-66.113,-177.620,7.666,148.770
C05116=1151.771,239.742,-66.139,-177.617,7.669,148.770
C05117=1151.767,239.990,-66.165,-177.615,7.671,148.770
C05118=1151.762,240.239,-66.192,-177.612,7.674,148.770
C05119=1151.758,240.487,-66.219,-177.609,7.677,148.770
C05120=1151.754,240.735,-66.246,-177.606,7.680,148.770
C05121=1151.749,240.984,-66.273,-177.604,7.682,148.770
C05122=1151.745,241.233,-66.299,-177.601,7.685,148.770
C05123=1151.740,241.481,-66.326,-177.598,7.688,148.770
C05124=1151.736,241.730,-66.353,-177.595,7.691,148.770
C05125=1151.731,241.978,-66.380,-177.592,7.694,148.769
C05126=1151.727,242.226,-66.406,-177.590,7.697,148.769
C05127=1151.723,242.475,-66.434,-177.587,7.700,148.769
C05128=1151.718,242.724,-66.461,-177.585,7.702,148.769
C05129=1151.714,242.972,-66.487,-177.582,7.705,148.769
C05130=1151.710,243.221,-66.514,-177.579,7.707,148.769
C05131=1151.705,243.469,-66.542,-177.576,7.710,148.769
C05132=1151.700,243.718,-66.569,-177.573,7.713,148.769
C05133=1151.696,243.966,-66.595,-177.570,7.716,148.769
C05134=1151.692,244.214,-66.622,-177.568,7.719,148.769
C05135=1151.687,244.463,-66.649,-177.565,7.721,148.768
C05136=1151.683,244.712,-66.677,-177.563,7.724,148.768
C05137=1151.679,244.960,-66.703,-177.560,7.727,148.768
C05138=1151.675,245.209,-66.730,-177.557,7.730,148.768
C05139=1151.670,245.457,-66.757,-177.554,7.733,148.768
C05140=1151.665,245.706,-66.784,-177.551,7.736,148.768
C05141=1151.661,245.954,-66.811,-177.549,7.739,148.768
C05142=1151.656,246.203,-66.838,-177.545,7.741,148.768
C05143=1151.653,246.452,-66.865,-177.543,7.743,148.768
C05144=1151.648,246.700,-66.892,-177.540,7.746,148.768
C05145=1151.644,246.948,-66.920,-177.538,7.749,148.767
C05146=1151.639,247.196,-66.947,-177.535,7.752,148.767
C05147=1151.634,247.445,-66.974,-177.532,7.755,148.767
C05148=1151.630,247.694,-67.002,-177.529,7.758,148.767
C05149=1151.626,247.943,-67.029,-177.527,7.761,148.767
C05150=1151.621,248.190,-67.056,-177.524,7.764,148.767
C05151=1151.617,248.439,-67.083,-177.521,7.767,148.767
C05152=1151.613,248.687,-67.110,-177.519,7.769,148.767
C05153=1151.609,248.936,-67.137,-177.516,7.772,148.767
C05154=1151.604,249.184,-67.165,-177.513,7.775,148.767
C05155=1151.600,249.433,-67.192,-177.510,7.778,148.767
C05156=1151.595,249.681,-67.219,-177.508,7.781,148.767
C05157=1151.591,249.930,-67.247,-177.505,7.784,148.767
C05158=1151.587,250.178,-67.274,-177.502,7.787,148.767
C05159=1151.582,250.427,-67.302,-177.499,7.790,148.766
C05160=1151.577,250.675,-67.329,-177.497,7.792,148.766
C05161=1151.573,250.924,-67.357,-177.494,7.795,148.766
C05162=1151.569,251.172,-67.384,-177.492,7.798,148.766
C05163=1151.564,251.420,-67.412,-177.489,7.800,148.766
C05164=1151.560,251.669,-67.439,-177.486,7.803,148.766
C05165=1151.556,251.917,-67.467,-177.483,7.806,148.766
C05166=1151.551,252.166,-67.494,-177.480,7.809,148.766
C05167=1151.547,252.414,-67.521,-177.478,7.812,148.766
C05168=1151.543,252.663,-67.549,-177.475,7.815,148.766
C05169=1151.538,252.911,-67.576,-177.472,7.818,148.766
C05170=1151.534,253.159,-67.604,-177.469,7.821,148.766
C05171=1151.529,253.409,-67.632,-177.467,7.824,148.766
C05172=1151.525,253.657,-67.660,-177.464,7.827,148.766
C05173=1151.520,253.905,-67.687,-177.461,7.830,148.765
C05174=1151.516,254.154,-67.715,-177.458,7.833,148.765
C05175=1151.512,254.402,-67.743,-177.456,7.835,148.765
C05176=1151.507,254.650,-67.770,-177.453,7.838,148.765
C05177=1151.504,254.899,-67.798,-177.450,7.841,148.765
C05178=1151.499,255.147,-67.825,-177.448,7.844,148.765
C05179=1151.494,255.395,-67.853,-177.445,7.847,148.765
C05180=1151.490,255.644,-67.881,-177.442,7.850,148.765
C05181=1151.485,255.892,-67.909,-177.439,7.852,148.765
C05182=1151.482,256.141,-67.937,-177.437,7.855,148.765
C05183=1151.477,256.389,-67.964,-177.434,7.858,148.765
C05184=1151.473,256.637,-67.991,-177.431,7.861,148.765
C05185=1151.468,256.886,-68.020,-177.428,7.864,148.765
C05186=1151.464,257.134,-68.048,-177.425,7.867,148.765
C05187=1151.459,257.383,-68.075,-177.423,7.870,148.765
C05188=1151.455,257.631,-68.103,-177.420,7.873,148.764
C05189=1151.450,257.879,-68.132,-177.417,7.876,148.764
C05190=1151.447,258.128,-68.160,-177.414,7.879,148.764
C05191=1151.442,258.376,-68.187,-177.412,7.882,148.764
C05192=1151.438,258.625,-68.215,-177.409,7.885,148.764
C05193=1151.433,258.873,-68.243,-177.406,7.888,148.764
C05194=1151.429,259.122,-68.271,-177.403,7.891,148.764
C05195=1151.425,259.370,-68.299,-177.402,7.893,148.764
C05196=1151.420,259.618,-68.327,-177.399,7.896,148.764
C05197=1151.416,259.867,-68.355,-177.396,7.899,148.764
C05198=1151.412,260.115,-68.383,-177.393,7.902,148.764
C05199=1151.407,260.364,-68.412,-177.390,7.905,148.764
C05200=1151.403,260.612,-68.439,-177.388,7.908,148.764
C05201=1151.399,260.860,-68.467,-177.385,7.911,148.764
C05202=1151.394,261.108,-68.496,-177.382,7.914,148.764
C05203=1151.389,261.382,-68.527,-177.379,7.917,148.764
C05204=1151.385,261.655,-68.557,-177.376,7.920,148.764
C05205=1151.380,261.928,-68.588,-177.373,7.923,148.764
C05206=1151.375,262.203,-68.619,-177.370,7.927,148.764
C05207=1151.371,262.451,-68.647,-177.367,7.930,148.764
C05208=1151.367,262.699,-68.675,-177.364,7.933,148.764
C05209=1151.362,262.947,-68.704,-177.361,7.936,148.763
C05210=1151.358,263.196,-68.732,-177.359,7.939,148.764
C05211=1151.353,263.444,-68.761,-177.356,7.942,148.764
C05212=1151.350,263.692,-68.789,-177.354,7.945,148.763
C05213=1151.345,263.940,-68.818,-177.351,7.948,148.763
C05214=1151.341,264.189,-68.846,-177.348,7.951,148.763
C05215=1151.336,264.437,-68.874,-177.345,7.954,148.763
C05216=1151.332,264.686,-68.902,-177.343,7.957,148.763
C05217=1151.327,264.934,-68.931,-177.340,7.960,148.763
C05218=1151.323,265.182,-68.959,-177.337,7.963,148.763
C05219=1151.319,265.431,-68.987,-177.335,7.966,148.763
C05220=1151.315,265.679,-69.016,-177.332,7.969,148.763
C05221=1151.310,265.927,-69.045,-177.329,7.972,148.763
C05222=1151.306,266.175,-69.072,-177.326,7.975,148.763
C05223=1151.301,266.424,-69.101,-177.324,7.978,148.763
C05224=1151.297,266.673,-69.129,-177.321,7.981,148.763
C05225=1151.293,266.920,-69.158,-177.318,7.984,148.763
C05226=1151.288,267.169,-69.187,-177.316,7.987,148.763
C05227=1151.284,267.417,-69.215,-177.313,7.990,148.763
C05228=1151.279,267.666,-69.244,-177.310,7.993,148.763
C05229=1151.276,267.914,-69.273,-177.307,7.996,148.763
C05230=1151.271,268.162,-69.301,-177.305,7.999,148.763
C05231=1151.266,268.411,-69.330,-177.302,8.002,148.763
C05232=1151.263,268.659,-69.359,-177.299,8.005,148.763
C05233=1151.258,268.907,-69.387,-177.297,8.008,148.763
C05234=1151.254,269.156,-69.415,-177.294,8.011,148.763
C05235=1151.250,269.404,-69.444,-177.291,8.014,148.763
C05236=1151.245,269.652,-69.473,-177.289,8.017,148.763
C05237=1151.241,269.900,-69.502,-177.286,8.020,148.763
C05238=1151.237,270.149,-69.530,-177.283,8.023,148.763
C05239=1151.232,270.397,-69.559,-177.281,8.026,148.763
C05240=1151.228,270.646,-69.588,-177.278,8.029,148.763
C05241=1151.224,270.894,-69.616,-177.275,8.032,148.763
C05242=1151.219,271.142,-69.645,-177.273,8.035,148.763
C05243=1151.215,271.391,-69.674,-177.270,8.038,148.763
C05244=1151.211,271.639,-69.703,-177.267,8.041,148.763
C05245=1151.207,271.887,-69.732,-177.264,8.044,148.763
C05246=1151.202,272.135,-69.761,-177.262,8.047,148.763
C05247=1151.197,272.384,-69.790,-177.259,8.050,148.763
C05248=1151.194,272.632,-69.819,-177.256,8.053,148.763
C05249=1151.189,272.881,-69.847,-177.253,8.057,148.763
C05250=1151.185,273.128,-69.876,-177.251,8.060,148.763
C05251=1151.181,273.377,-69.906,-177.248,8.063,148.763
C05252=1151.176,273.625,-69.935,-177.245,8.066,148.763
C05253=1151.173,273.873,-69.963,-177.242,8.069,148.763
C05254=1151.167,274.122,-69.992,-177.240,8.072,148.763
C05255=1151.163,274.370,-70.021,-177.237,8.075,148.763
C05256=1151.159,274.618,-70.051,-177.235,8.078,148.763
C05257=1151.155,274.867,-70.079,-177.232,8.081,148.763
C05258=1151.151,275.115,-70.108,-177.229,8.084,148.763
C05259=1151.146,275.363,-70.137,-177.227,8.087,148.763
C05260=1151.142,275.611,-70.167,-177.224,8.090,148.763
C05261=1151.138,275.860,-70.196,-177.221,8.093,148.763
C05262=1151.134,276.108,-70.225,-177.219,8.096,148.763
C05263=1151.129,276.356,-70.254,-177.216,8.099,148.763
C05264=1151.125,276.604,-70.284,-177.213,8.102,148.763
C05265=1151.120,276.853,-70.312,-177.210,8.106,148.763
C05266=1151.116,277.101,-70.342,-177.208,8.109,148.763
C05267=1151.112,277.349,-70.371,-177.205,8.112,148.763
C05268=1151.108,277.597,-70.400,-177.202,8.115,148.763
C05269=1151.104,277.845,-70.429,-177.199,8.118,148.763
C05270=1151.100,278.094,-70.458,-177.197,8.121,148.763
C05271=1151.095,278.342,-70.487,-177.194,8.124,148.763
C05272=1151.091,278.590,-70.517,-177.191,8.127,148.763
C05273=1151.086,278.838,-70.546,-177.189,8.130,148.763
C05274=1151.082,279.087,-70.576,-177.186,8.133,148.763
C05275=1151.078,279.335,-70.605,-177.184,8.136,148.763
C05276=1151.074,279.583,-70.635,-177.181,8.139,148.763
C05277=1151.070,279.831,-70.664,-177.178,8.143,148.763
C05278=1151.066,280.080,-70.693,-177.175,8.146,148.763
C05279=1151.061,280.328,-70.723,-177.173,8.149,148.763
C05280=1151.057,280.576,-70.752,-177.170,8.152,148.763
C05281=1151.052,280.824,-70.781,-177.167,8.155,148.763
C05282=1151.048,281.072,-70.811,-177.165,8.158,148.763
C05283=1151.043,281.321,-70.841,-177.162,8.162,148.763
C05284=1151.039,281.569,-70.870,-177.159,8.164,148.763
C05285=1151.035,281.817,-70.900,-177.157,8.167,148.763
C05286=1151.031,282.065,-70.929,-177.154,8.171,148.763
C05287=1151.027,282.314,-70.959,-177.151,8.174,148.763
C05288=1151.022,282.562,-70.988,-177.149,8.178,148.763
C05289=1151.018,282.810,-71.018,-177.146,8.181,148.763
C05290=1151.014,283.059,-71.047,-177.143,8.184,148.763
C05291=1151.009,283.307,-71.078,-177.141,8.187,148.764
C05292=1151.005,283.555,-71.107,-177.138,8.190,148.764
C05293=1151.001,283.803,-71.137,-177.135,8.193,148.763
C05294=1150.997,284.051,-71.166,-177.133,8.196,148.764
C05295=1150.993,284.300,-71.196,-177.130,8.199,148.764
C05296=1150.989,284.548,-71.225,-177.127,8.203,148.764
C05297=1150.984,284.796,-71.256,-177.124,8.206,148.764
C05298=1150.980,285.044,-71.285,-177.122,8.209,148.764
C05299=1150.976,285.292,-71.315,-177.119,8.212,148.764
C05300=1150.971,285.541,-71.344,-177.117,8.215,148.764
C05301=1150.968,285.788,-71.374,-177.114,8.218,148.764
C05302=1150.963,286.037,-71.405,-177.112,8.221,148.764
C05303=1150.958,286.285,-71.434,-177.109,8.224,148.764
C05304=1150.955,286.533,-71.464,-177.106,8.228,148.764
C05305=1150.950,286.781,-71.494,-177.103,8.231,148.764
C05306=1150.945,287.030,-71.524,-177.100,8.234,148.764
C05307=1150.941,287.304,-71.557,-177.098,8.238,148.764
C05308=1150.936,287.580,-71.590,-177.095,8.241,148.764
C05309=1150.932,287.855,-71.623,-177.091,8.245,148.764
C05310=1150.927,288.130,-71.657,-177.089,8.248,148.764
C05311=1150.922,288.379,-71.687,-177.086,8.251,148.764
C05312=1150.918,288.626,-71.717,-177.083,8.255,148.765
C05313=1150.914,288.874,-71.746,-177.081,8.258,148.765
C05314=1150.909,289.123,-71.776,-177.078,8.261,148.764
C05315=1150.905,289.371,-71.806,-177.075,8.265,148.765
C05316=1150.902,289.620,-71.836,-177.073,8.268,148.765
C05317=1150.897,289.868,-71.867,-177.070,8.271,148.765
C05318=1150.893,290.116,-71.896,-177.068,8.274,148.765
C05319=1150.888,290.364,-71.927,-177.065,8.278,148.765
C05320=1150.885,290.612,-71.957,-177.062,8.281,148.765
C05321=1150.880,290.860,-71.987,-177.060,8.284,148.765
C05322=1150.876,291.108,-72.018,-177.057,8.287,148.765
C05323=1150.872,291.357,-72.047,-177.055,8.290,148.765
C05324=1150.868,291.605,-72.078,-177.052,8.293,148.765
C05325=1150.863,291.853,-72.108,-177.048,8.297,148.765
C05326=1150.859,292.101,-72.138,-177.046,8.300,148.765
C05327=1150.855,292.349,-72.169,-177.043,8.303,148.765
C05328=1150.850,292.597,-72.199,-177.041,8.306,148.765
C05329=1150.847,292.845,-72.229,-177.038,8.309,148.765
C05330=1150.843,293.093,-72.259,-177.036,8.313,148.766
C05331=1150.838,293.341,-72.290,-177.033,8.316,148.766
C05332=1150.834,293.589,-72.320,-177.030,8.320,148.766
C05333=1150.829,293.837,-72.350,-177.027,8.323,148.766
C05334=1150.825,294.086,-72.381,-177.025,8.326,148.766
C05335=1150.821,294.334,-72.411,-177.022,8.329,148.766
C05336=1150.817,294.582,-72.442,-177.020,8.332,148.766
C05337=1150.813,294.830,-72.472,-177.017,8.336,148.766
C05338=1150.808,295.078,-72.503,-177.014,8.339,148.766
C05339=1150.805,295.326,-72.533,-177.012,8.342,148.766
C05340=1150.800,295.575,-72.563,-177.009,8.345,148.766
C05341=1150.796,295.822,-72.593,-177.007,8.348,148.766
C05342=1150.791,296.070,-72.624,-177.004,8.352,148.767
C05343=1150.787,296.319,-72.655,-177.001,8.355,148.767
C05344=1150.784,296.567,-72.685,-176.999,8.359,148.767
C05345=1150.779,296.815,-72.716,-176.996,8.362,148.767
C05346=1150.775,297.062,-72.746,-176.993,8.365,148.767
C05347=1150.771,297.311,-72.778,-176.991,8.369,148.767
C05348=1150.766,297.559,-72.808,-176.988,8.372,148.767
C05349=1150.763,297.806,-72.838,-176.985,8.375,148.767
C05350=1150.759,298.055,-72.870,-176.983,8.378,148.767
C05351=1150.754,298.303,-72.900,-176.980,8.381,148.767
C05352=1150.750,298.551,-72.931,-176.977,8.385,148.767
C05353=1150.746,298.799,-72.962,-176.975,8.388,148.768
C05354=1150.741,299.047,-72.992,-176.972,8.392,148.768
C05355=1150.737,299.295,-73.023,-176.970,8.395,148.768
C05356=1150.733,299.543,-73.053,-176.967,8.398,148.768
C05357=1150.729,299.792,-73.084,-176.964,8.402,148.768
C05358=1150.724,300.040,-73.115,-176.962,8.405,148.768
C05359=1150.720,300.288,-73.146,-176.959,8.408,148.768
C05360=1150.716,300.536,-73.177,-176.957,8.411,148.768
C05361=1150.712,300.784,-73.207,-176.954,8.414,148.768
C05362=1150.708,301.033,-73.238,-176.951,8.418,148.768
C05363=1150.703,301.280,-73.269,-176.949,8.421,148.769
C05364=1150.700,301.527,-73.300,-176.946,8.424,148.769
C05365=1150.696,301.776,-73.331,-176.943,8.428,148.769
C05366=1150.691,302.024,-73.362,-176.941,8.432,148.769
C05367=1150.686,302.272,-73.393,-176.938,8.435,148.769
C05368=1150.682,302.521,-73.424,-176.935,8.438,148.769
C05369=1150.678,302.768,-73.455,-176.933,8.441,148.769
C05370=1150.675,303.016,-73.486,-176.930,8.445,148.769
C05371=1150.670,303.264,-73.517,-176.927,8.448,148.769
C05372=1150.666,303.512,-73.547,-176.925,8.451,148.769
C05373=1150.662,303.760,-73.579,-176.922,8.455,148.770
C05374=1150.657,304.008,-73.610,-176.920,8.458,148.770
C05375=1150.653,304.257,-73.641,-176.917,8.462,148.770
C05376=1150.649,304.504,-73.673,-176.914,8.465,148.770
C05377=1150.644,304.752,-73.703,-176.912,8.468,148.770
C05378=1150.640,305.001,-73.735,-176.909,8.471,148.770
C05379=1150.636,305.248,-73.766,-176.906,8.475,148.770
C05380=1150.632,305.497,-73.797,-176.904,8.478,148.771
C05381=1150.627,305.745,-73.828,-176.901,8.481,148.770
C05382=1150.624,305.993,-73.859,-176.899,8.485,148.771
C05383=1150.620,306.241,-73.890,-176.896,8.489,148.771
C05384=1150.616,306.489,-73.922,-176.893,8.492,148.771
C05385=1150.611,306.737,-73.953,-176.891,8.495,148.771
C05386=1150.608,306.985,-73.984,-176.889,8.498,148.771
C05387=1150.603,307.233,-74.015,-176.885,8.502,148.771
C05388=1150.599,307.480,-74.047,-176.883,8.505,148.771
C05389=1150.595,307.729,-74.078,-176.881,8.509,148.772
C05390=1150.590,307.976,-74.110,-176.877,8.512,148.772
C05391=1150.586,308.225,-74.141,-176.875,8.516,148.772
C05392=1150.582,308.473,-74.173,-176.873,8.519,148.772
C05393=1150.577,308.721,-74.204,-176.870,8.522,148.772
C05394=1150.574,308.969,-74.235,-176.867,8.526,148.772
C05395=1150.569,309.217,-74.266,-176.865,8.529,148.772
C05396=1150.565,309.465,-74.298,-176.862,8.532,148.773
C05397=1150.561,309.712,-74.329,-176.860,8.535,148.773
C05398=1150.557,309.961,-74.361,-176.857,8.540,148.773
C05399=1150.553,310.208,-74.392,-176.854,8.543,148.773
C05400=1150.549,310.456,-74.424,-176.852,8.546,148.773
C05401=1150.544,310.704,-74.455,-176.849,8.550,148.773
C05402=1150.540,310.953,-74.487,-176.846,8.553,148.773
C05403=1150.536,311.201,-74.519,-176.844,8.556,148.773
C05404=1150.532,311.448,-74.550,-176.841,8.559,148.773
C05405=1150.528,311.697,-74.582,-176.838,8.563,148.774
C05406=1150.524,311.944,-74.613,-176.836,8.567,148.774
C05407=1150.520,312.192,-74.645,-176.834,8.570,148.774
C05408=1150.516,312.440,-74.677,-176.830,8.574,148.774
C05409=1150.511,312.688,-74.708,-176.828,8.577,148.774
C05410=1150.507,312.936,-74.740,-176.826,8.580,148.774
C05411=1150.503,313.214,-74.776,-176.823,8.584,148.775
C05412=1150.498,313.491,-74.811,-176.820,8.588,148.775
C05413=1150.493,313.769,-74.847,-176.817,8.592,148.775
C05414=1150.489,314.046,-74.883,-176.814,8.595,148.775
C05415=1150.485,314.295,-74.914,-176.811,8.600,148.775
C05416=1150.480,314.542,-74.945,-176.809,8.603,148.776
C05417=1150.476,314.790,-74.978,-176.806,8.606,148.776
C05418=1150.472,315.038,-75.010,-176.803,8.610,148.776
C05419=1150.468,315.286,-75.041,-176.801,8.613,148.776
C05420=1150.464,315.534,-75.073,-176.799,8.616,148.776
C05421=1150.460,315.782,-75.105,-176.796,8.621,148.776
C05422=1150.455,316.030,-75.137,-176.793,8.623,148.776
C05423=1150.452,316.278,-75.169,-176.791,8.627,148.777
C05424=1150.447,316.526,-75.201,-176.788,8.631,148.777
C05425=1150.443,316.773,-75.233,-176.786,8.634,148.777
C05426=1150.439,317.021,-75.264,-176.783,8.637,148.777
C05427=1150.435,317.270,-75.297,-176.780,8.641,148.777
C05428=1150.431,317.518,-75.329,-176.778,8.644,148.777
C05429=1150.427,317.765,-75.360,-176.775,8.648,148.778
C05430=1150.422,318.013,-75.393,-176.772,8.652,148.778
C05431=1150.419,318.261,-75.425,-176.770,8.655,148.778
C05432=1150.414,318.508,-75.457,-176.768,8.658,148.778
C05433=1150.410,318.756,-75.489,-176.765,8.661,148.778
C05434=1150.406,319.005,-75.521,-176.762,8.665,148.778
C05435=1150.402,319.253,-75.553,-176.760,8.669,148.779
C05436=1150.398,319.501,-75.585,-176.757,8.673,148.779
C05437=1150.394,319.748,-75.618,-176.755,8.676,148.779
C05438=1150.390,319.996,-75.650,-176.752,8.679,148.779
C05439=1150.385,320.244,-75.682,-176.749,8.683,148.779
C05440=1150.382,320.492,-75.714,-176.747,8.687,148.780
C05441=1150.377,320.739,-75.747,-176.744,8.690,148.780
C05442=1150.373,320.987,-75.779,-176.741,8.694,148.780
C05443=1150.369,321.236,-75.811,-176.739,8.697,148.780
C05444=1150.365,321.484,-75.843,-176.737,8.700,148.780
C05445=1150.361,321.732,-75.876,-176.734,8.704,148.780
C05446=1150.357,321.979,-75.908,-176.731,8.708,148.781
C05447=1150.352,322.227,-75.940,-176.729,8.711,148.781
C05448=1150.349,322.475,-75.973,-176.726,8.715,148.781
C05449=1150.344,322.723,-76.005,-176.724,8.718,148.781
C05450=1150.341,322.970,-76.038,-176.721,8.721,148.781
C05451=1150.337,323.219,-76.070,-176.718,8.725,148.781
C05452=1150.333,323.467,-76.102,-176.716,8.729,148.782
C05453=1150.328,323.714,-76.135,-176.713,8.733,148.782
C05454=1150.324,323.962,-76.167,-176.711,8.736,148.782
C05455=1150.320,324.210,-76.200,-176.708,8.739,148.782
C05456=1150.316,324.458,-76.232,-176.706,8.743,148.782
C05457=1150.312,324.705,-76.265,-176.703,8.747,148.783
C05458=1150.308,324.954,-76.297,-176.701,8.750,148.783
C05459=1150.304,325.201,-76.330,-176.698,8.754,148.783
C05460=1150.300,325.449,-76.362,-176.696,8.757,148.783
C05461=1150.295,325.697,-76.395,-176.693,8.761,148.784
C05462=1150.291,325.945,-76.427,-176.690,8.765,148.784
C05463=1150.288,326.192,-76.460,-176.688,8.768,148.784
C05464=1150.283,326.440,-76.493,-176.685,8.772,148.784
C05465=1150.279,326.688,-76.526,-176.683,8.775,148.784
C05466=1150.276,326.936,-76.558,-176.681,8.778,148.785
C05467=1150.271,327.184,-76.591,-176.678,8.783,148.785
C05468=1150.267,327.432,-76.624,-176.675,8.786,148.785
C05469=1150.263,327.680,-76.657,-176.672,8.790,148.785
C05470=1150.259,327.928,-76.689,-176.670,8.793,148.785
C05471=1150.255,328.175,-76.722,-176.667,8.796,148.785
C05472=1150.251,328.423,-76.755,-176.664,8.800,148.786
C05473=1150.246,328.671,-76.787,-176.662,8.803,148.786
C05474=1150.243,328.919,-76.820,-176.659,8.808,148.786
C05475=1150.239,329.167,-76.853,-176.657,8.811,148.786
C05476=1150.235,329.414,-76.886,-176.655,8.814,148.786
C05477=1150.230,329.663,-76.919,-176.652,8.818,148.787
C05478=1150.226,329.910,-76.952,-176.650,8.822,148.787
C05479=1150.223,330.158,-76.985,-176.647,8.826,148.787
C05480=1150.219,330.406,-77.018,-176.645,8.829,148.788
C05481=1150.214,330.653,-77.051,-176.642,8.832,148.788
C05482=1150.210,330.901,-77.084,-176.639,8.836,148.788
